(* IEC 61131-3 sources: Simulated-machine/integrations/openplc/thermal-plant-v4/pous/programs, 1 file *)

(* ---- main.st ---- *)
(* Generated by tools/generate_openplc_gateway.py.
   Raw Modbus values are intentionally retained; engineering_value = raw / scale.
   The cyclic task interval is 20 ms. *)
PROGRAM main
  VAR
    i_watchdog_scan_count : UINT := 0;
    i_watchdog_tick : BOOL := FALSE;
    i_condenser_last_echo : UINT := 0;
    i_condenser_echo_stale_ticks : UINT := 0;
    i_condenser_comm_lost : BOOL := FALSE;
    i_condensate_pump_last_echo : UINT := 0;
    i_condensate_pump_echo_stale_ticks : UINT := 0;
    i_condensate_pump_comm_lost : BOOL := FALSE;
    i_feedwater_tank_last_echo : UINT := 0;
    i_feedwater_tank_echo_stale_ticks : UINT := 0;
    i_feedwater_tank_comm_lost : BOOL := FALSE;
    i_feedwater_pump_last_echo : UINT := 0;
    i_feedwater_pump_echo_stale_ticks : UINT := 0;
    i_feedwater_pump_comm_lost : BOOL := FALSE;
    i_boiler_last_echo : UINT := 0;
    i_boiler_echo_stale_ticks : UINT := 0;
    i_boiler_comm_lost : BOOL := FALSE;
    i_steam_valve_last_echo : UINT := 0;
    i_steam_valve_echo_stale_ticks : UINT := 0;
    i_steam_valve_comm_lost : BOOL := FALSE;
    i_turbine_last_echo : UINT := 0;
    i_turbine_echo_stale_ticks : UINT := 0;
    i_turbine_comm_lost : BOOL := FALSE;
    i_generator_last_echo : UINT := 0;
    i_generator_echo_stale_ticks : UINT := 0;
    i_generator_comm_lost : BOOL := FALSE;
    i_condenser_start_active : BOOL := FALSE;
    i_condenser_start_scans : UINT := 0;
    i_condenser_stop_active : BOOL := FALSE;
    i_condenser_stop_scans : UINT := 0;
    i_condenser_reset_trip_active : BOOL := FALSE;
    i_condenser_reset_trip_scans : UINT := 0;
    i_condenser_ack_alarm_active : BOOL := FALSE;
    i_condenser_ack_alarm_scans : UINT := 0;
    i_condenser_trip_test_active : BOOL := FALSE;
    i_condenser_trip_test_scans : UINT := 0;
    i_condenser_clear_totalizer_active : BOOL := FALSE;
    i_condenser_clear_totalizer_scans : UINT := 0;
    i_condensate_pump_start_active : BOOL := FALSE;
    i_condensate_pump_start_scans : UINT := 0;
    i_condensate_pump_stop_active : BOOL := FALSE;
    i_condensate_pump_stop_scans : UINT := 0;
    i_condensate_pump_reset_trip_active : BOOL := FALSE;
    i_condensate_pump_reset_trip_scans : UINT := 0;
    i_condensate_pump_ack_alarm_active : BOOL := FALSE;
    i_condensate_pump_ack_alarm_scans : UINT := 0;
    i_condensate_pump_trip_test_active : BOOL := FALSE;
    i_condensate_pump_trip_test_scans : UINT := 0;
    i_condensate_pump_clear_totalizer_active : BOOL := FALSE;
    i_condensate_pump_clear_totalizer_scans : UINT := 0;
    i_feedwater_tank_start_active : BOOL := FALSE;
    i_feedwater_tank_start_scans : UINT := 0;
    i_feedwater_tank_stop_active : BOOL := FALSE;
    i_feedwater_tank_stop_scans : UINT := 0;
    i_feedwater_tank_reset_trip_active : BOOL := FALSE;
    i_feedwater_tank_reset_trip_scans : UINT := 0;
    i_feedwater_tank_ack_alarm_active : BOOL := FALSE;
    i_feedwater_tank_ack_alarm_scans : UINT := 0;
    i_feedwater_tank_trip_test_active : BOOL := FALSE;
    i_feedwater_tank_trip_test_scans : UINT := 0;
    i_feedwater_tank_clear_totalizer_active : BOOL := FALSE;
    i_feedwater_tank_clear_totalizer_scans : UINT := 0;
    i_feedwater_pump_start_active : BOOL := FALSE;
    i_feedwater_pump_start_scans : UINT := 0;
    i_feedwater_pump_stop_active : BOOL := FALSE;
    i_feedwater_pump_stop_scans : UINT := 0;
    i_feedwater_pump_reset_trip_active : BOOL := FALSE;
    i_feedwater_pump_reset_trip_scans : UINT := 0;
    i_feedwater_pump_ack_alarm_active : BOOL := FALSE;
    i_feedwater_pump_ack_alarm_scans : UINT := 0;
    i_feedwater_pump_trip_test_active : BOOL := FALSE;
    i_feedwater_pump_trip_test_scans : UINT := 0;
    i_feedwater_pump_clear_totalizer_active : BOOL := FALSE;
    i_feedwater_pump_clear_totalizer_scans : UINT := 0;
    i_boiler_start_active : BOOL := FALSE;
    i_boiler_start_scans : UINT := 0;
    i_boiler_stop_active : BOOL := FALSE;
    i_boiler_stop_scans : UINT := 0;
    i_boiler_reset_trip_active : BOOL := FALSE;
    i_boiler_reset_trip_scans : UINT := 0;
    i_boiler_ack_alarm_active : BOOL := FALSE;
    i_boiler_ack_alarm_scans : UINT := 0;
    i_boiler_trip_test_active : BOOL := FALSE;
    i_boiler_trip_test_scans : UINT := 0;
    i_boiler_clear_totalizer_active : BOOL := FALSE;
    i_boiler_clear_totalizer_scans : UINT := 0;
    i_steam_valve_start_active : BOOL := FALSE;
    i_steam_valve_start_scans : UINT := 0;
    i_steam_valve_stop_active : BOOL := FALSE;
    i_steam_valve_stop_scans : UINT := 0;
    i_steam_valve_reset_trip_active : BOOL := FALSE;
    i_steam_valve_reset_trip_scans : UINT := 0;
    i_steam_valve_ack_alarm_active : BOOL := FALSE;
    i_steam_valve_ack_alarm_scans : UINT := 0;
    i_steam_valve_trip_test_active : BOOL := FALSE;
    i_steam_valve_trip_test_scans : UINT := 0;
    i_steam_valve_clear_totalizer_active : BOOL := FALSE;
    i_steam_valve_clear_totalizer_scans : UINT := 0;
    i_turbine_start_active : BOOL := FALSE;
    i_turbine_start_scans : UINT := 0;
    i_turbine_stop_active : BOOL := FALSE;
    i_turbine_stop_scans : UINT := 0;
    i_turbine_reset_trip_active : BOOL := FALSE;
    i_turbine_reset_trip_scans : UINT := 0;
    i_turbine_ack_alarm_active : BOOL := FALSE;
    i_turbine_ack_alarm_scans : UINT := 0;
    i_turbine_trip_test_active : BOOL := FALSE;
    i_turbine_trip_test_scans : UINT := 0;
    i_turbine_clear_totalizer_active : BOOL := FALSE;
    i_turbine_clear_totalizer_scans : UINT := 0;
    i_generator_start_active : BOOL := FALSE;
    i_generator_start_scans : UINT := 0;
    i_generator_stop_active : BOOL := FALSE;
    i_generator_stop_scans : UINT := 0;
    i_generator_reset_trip_active : BOOL := FALSE;
    i_generator_reset_trip_scans : UINT := 0;
    i_generator_ack_alarm_active : BOOL := FALSE;
    i_generator_ack_alarm_scans : UINT := 0;
    i_generator_trip_test_active : BOOL := FALSE;
    i_generator_trip_test_scans : UINT := 0;
    i_generator_clear_totalizer_active : BOOL := FALSE;
    i_generator_clear_totalizer_scans : UINT := 0;
    i_generator_breaker_close_active : BOOL := FALSE;
    i_generator_breaker_close_scans : UINT := 0;
    i_generator_breaker_open_active : BOOL := FALSE;
    i_generator_breaker_open_scans : UINT := 0;
    i_turbine_trip_prev : BOOL := FALSE;
    i_boiler_trip_prev : BOOL := FALSE;
    i_condenser_trip_prev : BOOL := FALSE;
    i_feedwater_pump_trip_prev : BOOL := FALSE;
    i_condensate_pump_trip_prev : BOOL := FALSE;
    i_steam_valve_trip_prev : BOOL := FALSE;

    (* Southbound mirrors and commands.  Aliases match remote JSON exactly. *)
    condenser__input__status_word AT %IW0 : UINT := 0;
    condenser__input__alarm_word_1 AT %IW1 : UINT := 0;
    condenser__input__alarm_word_2 AT %IW2 : UINT := 0;
    condenser__input__trip_word AT %IW3 : UINT := 0;
    condenser__input__device_state AT %IW4 : UINT := 0;
    condenser__input__first_out_code AT %IW5 : UINT := 0;
    condenser__input__overall_quality AT %IW6 : UINT := 0;
    condenser__input__register_map_version AT %IW7 : UINT := 0;
    condenser__input__firmware_version AT %IW8 : UINT := 0;
    condenser__input__condenser_pressure AT %IW9 : UINT := 0;
    condenser__input__vacuum AT %IW10 : UINT := 0;
    condenser__input__hotwell_level AT %IW11 : UINT := 0;
    condenser__input__exhaust_inflow AT %IW12 : UINT := 0;
    condenser__input__condensing_capacity AT %IW13 : UINT := 0;
    condenser__input__actual_condensed AT %IW14 : UINT := 0;
    condenser__input__condensate_outflow AT %IW15 : UINT := 0;
    condenser__input__cooling_water_availability AT %IW16 : UINT := 0;
    condenser__input__vacuum_system_output AT %IW17 : UINT := 0;
    condenser__input__condensate_temperature AT %IW18 : UINT := 0;
    condenser__input__hotwell_mass_hi AT %IW19 : UINT := 0;
    condenser__input__hotwell_mass_lo AT %IW20 : UINT := 0;
    condenser__input__reserved_21 AT %IW21 : UINT := 0;
    condenser__input__reserved_22 AT %IW22 : UINT := 0;
    condenser__input__reserved_23 AT %IW23 : UINT := 0;
    condenser__input__reserved_24 AT %IW24 : UINT := 0;
    condenser__input__reserved_25 AT %IW25 : UINT := 0;
    condenser__input__reserved_26 AT %IW26 : UINT := 0;
    condenser__input__reserved_27 AT %IW27 : UINT := 0;
    condenser__input__reserved_28 AT %IW28 : UINT := 0;
    condenser__input__watchdog_echo AT %IW29 : UINT := 0;
    condenser__input__scan_time_ms AT %IW30 : UINT := 0;
    condenser__input__modbus_request_count AT %IW31 : UINT := 0;
    condenser__input__rejected_command_count AT %IW32 : UINT := 0;
    condenser__input__exception_count AT %IW33 : UINT := 0;
    condenser__input__sim_quality_word AT %IW34 : UINT := 0;
    condenser__input__sim_tick_low AT %IW35 : UINT := 0;
    condenser__input__comm_loss_seconds AT %IW36 : UINT := 0;
    condenser__input__fault_inject_word AT %IW37 : UINT := 0;
    condenser__input__snapshot_generation AT %IW38 : UINT := 0;
    condenser__input__run_seconds_hi AT %IW39 : UINT := 0;
    condenser__input__run_seconds_lo AT %IW40 : UINT := 0;
    condenser__input__start_count AT %IW41 : UINT := 0;
    condenser__input__trip_count AT %IW42 : UINT := 0;
    condenser__input__mass_total_hi AT %IW43 : UINT := 0;
    condenser__input__mass_total_lo AT %IW44 : UINT := 0;
    condenser__input__energy_total_hi AT %IW45 : UINT := 0;
    condenser__input__energy_total_lo AT %IW46 : UINT := 0;
    condenser__input__alarm_count AT %IW47 : UINT := 0;
    condenser__input__accepted_command_count AT %IW48 : UINT := 0;
    condenser__input__reserved_49 AT %IW49 : UINT := 0;
    condenser__discrete__ready AT %IX0.0 : BOOL := FALSE;
    condenser__discrete__running AT %IX0.1 : BOOL := FALSE;
    condenser__discrete__starting AT %IX0.2 : BOOL := FALSE;
    condenser__discrete__stopping AT %IX0.3 : BOOL := FALSE;
    condenser__discrete__tripped AT %IX0.4 : BOOL := FALSE;
    condenser__discrete__alarm_active AT %IX0.5 : BOOL := FALSE;
    condenser__discrete__local_mode AT %IX0.6 : BOOL := FALSE;
    condenser__discrete__remote_mode AT %IX0.7 : BOOL := FALSE;
    condenser__discrete__auto_mode AT %IX1.0 : BOOL := FALSE;
    condenser__discrete__manual_mode AT %IX1.1 : BOOL := FALSE;
    condenser__discrete__control_watchdog_ok AT %IX1.2 : BOOL := FALSE;
    condenser__discrete__sim_bus_ok AT %IX1.3 : BOOL := FALSE;
    condenser__discrete__interlocks_ok AT %IX1.4 : BOOL := FALSE;
    condenser__discrete__sensor_fault AT %IX1.5 : BOOL := FALSE;
    condenser__discrete__actuator_fault AT %IX1.6 : BOOL := FALSE;
    condenser__discrete__maintenance_mode AT %IX1.7 : BOOL := FALSE;
    condenser__holding_readback__control_mode AT %IW512 : UINT := 0;
    condenser__holding_readback__command_sequence AT %IW513 : UINT := 0;
    condenser__holding_readback__watchdog_counter AT %IW514 : UINT := 0;
    condenser__holding_readback__reset_key AT %IW515 : UINT := 0;
    condenser__holding_readback__simulation_flags AT %IW516 : UINT := 0;
    condenser__holding_readback__active_controller_id AT %IW517 : UINT := 0;
    condenser__holding_readback__command_lease_time AT %IW518 : UINT := 0;
    condenser__holding_readback__output_rate_limit AT %IW519 : UINT := 0;
    condenser__holding_readback__reserved AT %IW520 : UINT := 0;
    condenser__holding_readback__primary_setpoint AT %IW521 : UINT := 0;
    condenser__holding_readback__secondary_setpoint AT %IW522 : UINT := 0;
    condenser__holding_readback__manual_output AT %IW523 : UINT := 0;
    condenser__holding_readback__output_high_limit AT %IW524 : UINT := 0;
    condenser__holding_readback__output_low_limit AT %IW525 : UINT := 0;
    condenser__holding_readback__reserved_14 AT %IW526 : UINT := 0;
    condenser__holding_readback__reserved_15 AT %IW527 : UINT := 0;
    condenser__holding_readback__reserved_16 AT %IW528 : UINT := 0;
    condenser__holding_readback__reserved_17 AT %IW529 : UINT := 0;
    condenser__holding_readback__reserved_18 AT %IW530 : UINT := 0;
    condenser__holding_readback__pid_kp AT %IW531 : UINT := 0;
    condenser__holding_readback__pid_ki AT %IW532 : UINT := 0;
    condenser__holding_readback__pid_kd AT %IW533 : UINT := 0;
    condenser__holding_readback__deadband AT %IW534 : UINT := 0;
    condenser__holding_readback__integral_limit AT %IW535 : UINT := 0;
    condenser__holding_readback__controller_scan_time AT %IW536 : UINT := 0;
    condenser__holding_readback__reserved_25 AT %IW537 : UINT := 0;
    condenser__holding_readback__reserved_26 AT %IW538 : UINT := 0;
    condenser__holding_readback__reserved_27 AT %IW539 : UINT := 0;
    condenser__holding_readback__reserved_28 AT %IW540 : UINT := 0;
    condenser__holding_readback__makeup_valve_cmd AT %IW541 : UINT := 0;
    condenser__holding_readback__reserved_30 AT %IW542 : UINT := 0;
    condenser__holding_readback__reserved_31 AT %IW543 : UINT := 0;
    condenser__coil__start AT %QX0.0 : BOOL := FALSE;
    condenser__coil__stop AT %QX0.1 : BOOL := FALSE;
    condenser__coil__reset_trip AT %QX0.2 : BOOL := FALSE;
    condenser__coil__ack_alarm AT %QX0.3 : BOOL := FALSE;
    condenser__coil__emergency_stop AT %QX0.4 : BOOL := FALSE;
    condenser__coil__force_safe AT %QX0.5 : BOOL := FALSE;
    condenser__coil__trip_test AT %QX0.6 : BOOL := FALSE;
    condenser__coil__clear_totalizer AT %QX0.7 : BOOL := FALSE;
    condenser__holding__control_mode AT %QW0 : UINT := 3;
    condenser__holding__command_sequence AT %QW1 : UINT := 0;
    condenser__holding__watchdog_counter AT %QW2 : UINT := 1;
    condenser__holding__reset_key AT %QW3 : UINT := 0;
    condenser__holding__simulation_flags AT %QW4 : UINT := 0;
    condenser__holding__active_controller_id AT %QW5 : UINT := 1;
    condenser__holding__command_lease_time AT %QW6 : UINT := 5;
    condenser__holding__output_rate_limit AT %QW7 : UINT := 1000;
    condenser__holding__reserved AT %QW8 : UINT := 0;
    condenser__holding__primary_setpoint AT %QW9 : UINT := 0;
    condenser__holding__secondary_setpoint AT %QW10 : UINT := 0;
    condenser__holding__manual_output AT %QW11 : UINT := 0;
    condenser__holding__output_high_limit AT %QW12 : UINT := 10000;
    condenser__holding__output_low_limit AT %QW13 : UINT := 0;
    condenser__holding__pid_kp AT %QW19 : UINT := 0;
    condenser__holding__pid_ki AT %QW20 : UINT := 0;
    condenser__holding__pid_kd AT %QW21 : UINT := 0;
    condenser__holding__deadband AT %QW22 : UINT := 0;
    condenser__holding__integral_limit AT %QW23 : UINT := 0;
    condenser__holding__controller_scan_time AT %QW24 : UINT := 200;
    condenser__holding__makeup_valve_cmd AT %QW29 : UINT := 0;
    condensate_pump__input__status_word AT %IW64 : UINT := 0;
    condensate_pump__input__alarm_word_1 AT %IW65 : UINT := 0;
    condensate_pump__input__alarm_word_2 AT %IW66 : UINT := 0;
    condensate_pump__input__trip_word AT %IW67 : UINT := 0;
    condensate_pump__input__device_state AT %IW68 : UINT := 0;
    condensate_pump__input__first_out_code AT %IW69 : UINT := 0;
    condensate_pump__input__overall_quality AT %IW70 : UINT := 0;
    condensate_pump__input__register_map_version AT %IW71 : UINT := 0;
    condensate_pump__input__firmware_version AT %IW72 : UINT := 0;
    condensate_pump__input__actual_speed AT %IW73 : UINT := 0;
    condensate_pump__input__flow AT %IW74 : UINT := 0;
    condensate_pump__input__suction_pressure AT %IW75 : UINT := 0;
    condensate_pump__input__discharge_pressure AT %IW76 : UINT := 0;
    condensate_pump__input__motor_current AT %IW77 : UINT := 0;
    condensate_pump__input__npsh_margin AT %IW78 : UINT := 0;
    condensate_pump__input__vibration AT %IW79 : UINT := 0;
    condensate_pump__input__source_level AT %IW80 : UINT := 0;
    condensate_pump__input__backpressure AT %IW81 : UINT := 0;
    condensate_pump__input__outlet_valve_position AT %IW82 : UINT := 0;
    condensate_pump__input__cavitation_factor AT %IW83 : UINT := 0;
    condensate_pump__input__reserved_20 AT %IW84 : UINT := 0;
    condensate_pump__input__reserved_21 AT %IW85 : UINT := 0;
    condensate_pump__input__reserved_22 AT %IW86 : UINT := 0;
    condensate_pump__input__reserved_23 AT %IW87 : UINT := 0;
    condensate_pump__input__reserved_24 AT %IW88 : UINT := 0;
    condensate_pump__input__reserved_25 AT %IW89 : UINT := 0;
    condensate_pump__input__reserved_26 AT %IW90 : UINT := 0;
    condensate_pump__input__reserved_27 AT %IW91 : UINT := 0;
    condensate_pump__input__reserved_28 AT %IW92 : UINT := 0;
    condensate_pump__input__watchdog_echo AT %IW93 : UINT := 0;
    condensate_pump__input__scan_time_ms AT %IW94 : UINT := 0;
    condensate_pump__input__modbus_request_count AT %IW95 : UINT := 0;
    condensate_pump__input__rejected_command_count AT %IW96 : UINT := 0;
    condensate_pump__input__exception_count AT %IW97 : UINT := 0;
    condensate_pump__input__sim_quality_word AT %IW98 : UINT := 0;
    condensate_pump__input__sim_tick_low AT %IW99 : UINT := 0;
    condensate_pump__input__comm_loss_seconds AT %IW100 : UINT := 0;
    condensate_pump__input__fault_inject_word AT %IW101 : UINT := 0;
    condensate_pump__input__snapshot_generation AT %IW102 : UINT := 0;
    condensate_pump__input__run_seconds_hi AT %IW103 : UINT := 0;
    condensate_pump__input__run_seconds_lo AT %IW104 : UINT := 0;
    condensate_pump__input__start_count AT %IW105 : UINT := 0;
    condensate_pump__input__trip_count AT %IW106 : UINT := 0;
    condensate_pump__input__mass_total_hi AT %IW107 : UINT := 0;
    condensate_pump__input__mass_total_lo AT %IW108 : UINT := 0;
    condensate_pump__input__energy_total_hi AT %IW109 : UINT := 0;
    condensate_pump__input__energy_total_lo AT %IW110 : UINT := 0;
    condensate_pump__input__alarm_count AT %IW111 : UINT := 0;
    condensate_pump__input__accepted_command_count AT %IW112 : UINT := 0;
    condensate_pump__input__reserved_49 AT %IW113 : UINT := 0;
    condensate_pump__discrete__ready AT %IX2.0 : BOOL := FALSE;
    condensate_pump__discrete__running AT %IX2.1 : BOOL := FALSE;
    condensate_pump__discrete__starting AT %IX2.2 : BOOL := FALSE;
    condensate_pump__discrete__stopping AT %IX2.3 : BOOL := FALSE;
    condensate_pump__discrete__tripped AT %IX2.4 : BOOL := FALSE;
    condensate_pump__discrete__alarm_active AT %IX2.5 : BOOL := FALSE;
    condensate_pump__discrete__local_mode AT %IX2.6 : BOOL := FALSE;
    condensate_pump__discrete__remote_mode AT %IX2.7 : BOOL := FALSE;
    condensate_pump__discrete__auto_mode AT %IX3.0 : BOOL := FALSE;
    condensate_pump__discrete__manual_mode AT %IX3.1 : BOOL := FALSE;
    condensate_pump__discrete__control_watchdog_ok AT %IX3.2 : BOOL := FALSE;
    condensate_pump__discrete__sim_bus_ok AT %IX3.3 : BOOL := FALSE;
    condensate_pump__discrete__interlocks_ok AT %IX3.4 : BOOL := FALSE;
    condensate_pump__discrete__sensor_fault AT %IX3.5 : BOOL := FALSE;
    condensate_pump__discrete__actuator_fault AT %IX3.6 : BOOL := FALSE;
    condensate_pump__discrete__maintenance_mode AT %IX3.7 : BOOL := FALSE;
    condensate_pump__holding_readback__control_mode AT %IW576 : UINT := 0;
    condensate_pump__holding_readback__command_sequence AT %IW577 : UINT := 0;
    condensate_pump__holding_readback__watchdog_counter AT %IW578 : UINT := 0;
    condensate_pump__holding_readback__reset_key AT %IW579 : UINT := 0;
    condensate_pump__holding_readback__simulation_flags AT %IW580 : UINT := 0;
    condensate_pump__holding_readback__active_controller_id AT %IW581 : UINT := 0;
    condensate_pump__holding_readback__command_lease_time AT %IW582 : UINT := 0;
    condensate_pump__holding_readback__output_rate_limit AT %IW583 : UINT := 0;
    condensate_pump__holding_readback__reserved AT %IW584 : UINT := 0;
    condensate_pump__holding_readback__primary_setpoint AT %IW585 : UINT := 0;
    condensate_pump__holding_readback__secondary_setpoint AT %IW586 : UINT := 0;
    condensate_pump__holding_readback__manual_output AT %IW587 : UINT := 0;
    condensate_pump__holding_readback__output_high_limit AT %IW588 : UINT := 0;
    condensate_pump__holding_readback__output_low_limit AT %IW589 : UINT := 0;
    condensate_pump__holding_readback__reserved_14 AT %IW590 : UINT := 0;
    condensate_pump__holding_readback__reserved_15 AT %IW591 : UINT := 0;
    condensate_pump__holding_readback__reserved_16 AT %IW592 : UINT := 0;
    condensate_pump__holding_readback__reserved_17 AT %IW593 : UINT := 0;
    condensate_pump__holding_readback__reserved_18 AT %IW594 : UINT := 0;
    condensate_pump__holding_readback__pid_kp AT %IW595 : UINT := 0;
    condensate_pump__holding_readback__pid_ki AT %IW596 : UINT := 0;
    condensate_pump__holding_readback__pid_kd AT %IW597 : UINT := 0;
    condensate_pump__holding_readback__deadband AT %IW598 : UINT := 0;
    condensate_pump__holding_readback__integral_limit AT %IW599 : UINT := 0;
    condensate_pump__holding_readback__controller_scan_time AT %IW600 : UINT := 0;
    condensate_pump__holding_readback__reserved_25 AT %IW601 : UINT := 0;
    condensate_pump__holding_readback__reserved_26 AT %IW602 : UINT := 0;
    condensate_pump__holding_readback__reserved_27 AT %IW603 : UINT := 0;
    condensate_pump__holding_readback__reserved_28 AT %IW604 : UINT := 0;
    condensate_pump__holding_readback__reserved_29 AT %IW605 : UINT := 0;
    condensate_pump__holding_readback__reserved_30 AT %IW606 : UINT := 0;
    condensate_pump__holding_readback__reserved_31 AT %IW607 : UINT := 0;
    condensate_pump__coil__start AT %QX2.0 : BOOL := FALSE;
    condensate_pump__coil__stop AT %QX2.1 : BOOL := FALSE;
    condensate_pump__coil__reset_trip AT %QX2.2 : BOOL := FALSE;
    condensate_pump__coil__ack_alarm AT %QX2.3 : BOOL := FALSE;
    condensate_pump__coil__emergency_stop AT %QX2.4 : BOOL := FALSE;
    condensate_pump__coil__force_safe AT %QX2.5 : BOOL := FALSE;
    condensate_pump__coil__trip_test AT %QX2.6 : BOOL := FALSE;
    condensate_pump__coil__clear_totalizer AT %QX2.7 : BOOL := FALSE;
    condensate_pump__holding__control_mode AT %QW64 : UINT := 3;
    condensate_pump__holding__command_sequence AT %QW65 : UINT := 0;
    condensate_pump__holding__watchdog_counter AT %QW66 : UINT := 1;
    condensate_pump__holding__reset_key AT %QW67 : UINT := 0;
    condensate_pump__holding__simulation_flags AT %QW68 : UINT := 0;
    condensate_pump__holding__active_controller_id AT %QW69 : UINT := 2;
    condensate_pump__holding__command_lease_time AT %QW70 : UINT := 5;
    condensate_pump__holding__output_rate_limit AT %QW71 : UINT := 1000;
    condensate_pump__holding__reserved AT %QW72 : UINT := 0;
    condensate_pump__holding__primary_setpoint AT %QW73 : UINT := 0;
    condensate_pump__holding__secondary_setpoint AT %QW74 : UINT := 0;
    condensate_pump__holding__manual_output AT %QW75 : UINT := 0;
    condensate_pump__holding__output_high_limit AT %QW76 : UINT := 10000;
    condensate_pump__holding__output_low_limit AT %QW77 : UINT := 0;
    condensate_pump__holding__pid_kp AT %QW83 : UINT := 0;
    condensate_pump__holding__pid_ki AT %QW84 : UINT := 0;
    condensate_pump__holding__pid_kd AT %QW85 : UINT := 0;
    condensate_pump__holding__deadband AT %QW86 : UINT := 0;
    condensate_pump__holding__integral_limit AT %QW87 : UINT := 0;
    condensate_pump__holding__controller_scan_time AT %QW88 : UINT := 200;
    feedwater_tank__input__status_word AT %IW128 : UINT := 0;
    feedwater_tank__input__alarm_word_1 AT %IW129 : UINT := 0;
    feedwater_tank__input__alarm_word_2 AT %IW130 : UINT := 0;
    feedwater_tank__input__trip_word AT %IW131 : UINT := 0;
    feedwater_tank__input__device_state AT %IW132 : UINT := 0;
    feedwater_tank__input__first_out_code AT %IW133 : UINT := 0;
    feedwater_tank__input__overall_quality AT %IW134 : UINT := 0;
    feedwater_tank__input__register_map_version AT %IW135 : UINT := 0;
    feedwater_tank__input__firmware_version AT %IW136 : UINT := 0;
    feedwater_tank__input__tank_level AT %IW137 : UINT := 0;
    feedwater_tank__input__tank_mass_hi AT %IW138 : UINT := 0;
    feedwater_tank__input__tank_mass_lo AT %IW139 : UINT := 0;
    feedwater_tank__input__condensate_inflow AT %IW140 : UINT := 0;
    feedwater_tank__input__feedwater_outflow AT %IW141 : UINT := 0;
    feedwater_tank__input__water_temperature AT %IW142 : UINT := 0;
    feedwater_tank__input__tank_pressure AT %IW143 : UINT := 0;
    feedwater_tank__input__overflow_flow AT %IW144 : UINT := 0;
    feedwater_tank__input__net_flow AT %IW145 : UINT := 0;
    feedwater_tank__input__reserved_18 AT %IW146 : UINT := 0;
    feedwater_tank__input__reserved_19 AT %IW147 : UINT := 0;
    feedwater_tank__input__reserved_20 AT %IW148 : UINT := 0;
    feedwater_tank__input__reserved_21 AT %IW149 : UINT := 0;
    feedwater_tank__input__reserved_22 AT %IW150 : UINT := 0;
    feedwater_tank__input__reserved_23 AT %IW151 : UINT := 0;
    feedwater_tank__input__reserved_24 AT %IW152 : UINT := 0;
    feedwater_tank__input__reserved_25 AT %IW153 : UINT := 0;
    feedwater_tank__input__reserved_26 AT %IW154 : UINT := 0;
    feedwater_tank__input__reserved_27 AT %IW155 : UINT := 0;
    feedwater_tank__input__reserved_28 AT %IW156 : UINT := 0;
    feedwater_tank__input__watchdog_echo AT %IW157 : UINT := 0;
    feedwater_tank__input__scan_time_ms AT %IW158 : UINT := 0;
    feedwater_tank__input__modbus_request_count AT %IW159 : UINT := 0;
    feedwater_tank__input__rejected_command_count AT %IW160 : UINT := 0;
    feedwater_tank__input__exception_count AT %IW161 : UINT := 0;
    feedwater_tank__input__sim_quality_word AT %IW162 : UINT := 0;
    feedwater_tank__input__sim_tick_low AT %IW163 : UINT := 0;
    feedwater_tank__input__comm_loss_seconds AT %IW164 : UINT := 0;
    feedwater_tank__input__fault_inject_word AT %IW165 : UINT := 0;
    feedwater_tank__input__snapshot_generation AT %IW166 : UINT := 0;
    feedwater_tank__input__run_seconds_hi AT %IW167 : UINT := 0;
    feedwater_tank__input__run_seconds_lo AT %IW168 : UINT := 0;
    feedwater_tank__input__start_count AT %IW169 : UINT := 0;
    feedwater_tank__input__trip_count AT %IW170 : UINT := 0;
    feedwater_tank__input__mass_total_hi AT %IW171 : UINT := 0;
    feedwater_tank__input__mass_total_lo AT %IW172 : UINT := 0;
    feedwater_tank__input__energy_total_hi AT %IW173 : UINT := 0;
    feedwater_tank__input__energy_total_lo AT %IW174 : UINT := 0;
    feedwater_tank__input__alarm_count AT %IW175 : UINT := 0;
    feedwater_tank__input__accepted_command_count AT %IW176 : UINT := 0;
    feedwater_tank__input__reserved_49 AT %IW177 : UINT := 0;
    feedwater_tank__discrete__ready AT %IX4.0 : BOOL := FALSE;
    feedwater_tank__discrete__running AT %IX4.1 : BOOL := FALSE;
    feedwater_tank__discrete__starting AT %IX4.2 : BOOL := FALSE;
    feedwater_tank__discrete__stopping AT %IX4.3 : BOOL := FALSE;
    feedwater_tank__discrete__tripped AT %IX4.4 : BOOL := FALSE;
    feedwater_tank__discrete__alarm_active AT %IX4.5 : BOOL := FALSE;
    feedwater_tank__discrete__local_mode AT %IX4.6 : BOOL := FALSE;
    feedwater_tank__discrete__remote_mode AT %IX4.7 : BOOL := FALSE;
    feedwater_tank__discrete__auto_mode AT %IX5.0 : BOOL := FALSE;
    feedwater_tank__discrete__manual_mode AT %IX5.1 : BOOL := FALSE;
    feedwater_tank__discrete__control_watchdog_ok AT %IX5.2 : BOOL := FALSE;
    feedwater_tank__discrete__sim_bus_ok AT %IX5.3 : BOOL := FALSE;
    feedwater_tank__discrete__interlocks_ok AT %IX5.4 : BOOL := FALSE;
    feedwater_tank__discrete__sensor_fault AT %IX5.5 : BOOL := FALSE;
    feedwater_tank__discrete__actuator_fault AT %IX5.6 : BOOL := FALSE;
    feedwater_tank__discrete__maintenance_mode AT %IX5.7 : BOOL := FALSE;
    feedwater_tank__holding_readback__control_mode AT %IW640 : UINT := 0;
    feedwater_tank__holding_readback__command_sequence AT %IW641 : UINT := 0;
    feedwater_tank__holding_readback__watchdog_counter AT %IW642 : UINT := 0;
    feedwater_tank__holding_readback__reset_key AT %IW643 : UINT := 0;
    feedwater_tank__holding_readback__simulation_flags AT %IW644 : UINT := 0;
    feedwater_tank__holding_readback__active_controller_id AT %IW645 : UINT := 0;
    feedwater_tank__holding_readback__command_lease_time AT %IW646 : UINT := 0;
    feedwater_tank__holding_readback__output_rate_limit AT %IW647 : UINT := 0;
    feedwater_tank__holding_readback__reserved AT %IW648 : UINT := 0;
    feedwater_tank__holding_readback__primary_setpoint AT %IW649 : UINT := 0;
    feedwater_tank__holding_readback__secondary_setpoint AT %IW650 : UINT := 0;
    feedwater_tank__holding_readback__manual_output AT %IW651 : UINT := 0;
    feedwater_tank__holding_readback__output_high_limit AT %IW652 : UINT := 0;
    feedwater_tank__holding_readback__output_low_limit AT %IW653 : UINT := 0;
    feedwater_tank__holding_readback__reserved_14 AT %IW654 : UINT := 0;
    feedwater_tank__holding_readback__reserved_15 AT %IW655 : UINT := 0;
    feedwater_tank__holding_readback__reserved_16 AT %IW656 : UINT := 0;
    feedwater_tank__holding_readback__reserved_17 AT %IW657 : UINT := 0;
    feedwater_tank__holding_readback__reserved_18 AT %IW658 : UINT := 0;
    feedwater_tank__holding_readback__pid_kp AT %IW659 : UINT := 0;
    feedwater_tank__holding_readback__pid_ki AT %IW660 : UINT := 0;
    feedwater_tank__holding_readback__pid_kd AT %IW661 : UINT := 0;
    feedwater_tank__holding_readback__deadband AT %IW662 : UINT := 0;
    feedwater_tank__holding_readback__integral_limit AT %IW663 : UINT := 0;
    feedwater_tank__holding_readback__controller_scan_time AT %IW664 : UINT := 0;
    feedwater_tank__holding_readback__reserved_25 AT %IW665 : UINT := 0;
    feedwater_tank__holding_readback__reserved_26 AT %IW666 : UINT := 0;
    feedwater_tank__holding_readback__reserved_27 AT %IW667 : UINT := 0;
    feedwater_tank__holding_readback__reserved_28 AT %IW668 : UINT := 0;
    feedwater_tank__holding_readback__heating_setpoint AT %IW669 : UINT := 0;
    feedwater_tank__holding_readback__reserved_30 AT %IW670 : UINT := 0;
    feedwater_tank__holding_readback__reserved_31 AT %IW671 : UINT := 0;
    feedwater_tank__coil__start AT %QX4.0 : BOOL := FALSE;
    feedwater_tank__coil__stop AT %QX4.1 : BOOL := FALSE;
    feedwater_tank__coil__reset_trip AT %QX4.2 : BOOL := FALSE;
    feedwater_tank__coil__ack_alarm AT %QX4.3 : BOOL := FALSE;
    feedwater_tank__coil__emergency_stop AT %QX4.4 : BOOL := FALSE;
    feedwater_tank__coil__force_safe AT %QX4.5 : BOOL := FALSE;
    feedwater_tank__coil__trip_test AT %QX4.6 : BOOL := FALSE;
    feedwater_tank__coil__clear_totalizer AT %QX4.7 : BOOL := FALSE;
    feedwater_tank__holding__control_mode AT %QW128 : UINT := 3;
    feedwater_tank__holding__command_sequence AT %QW129 : UINT := 0;
    feedwater_tank__holding__watchdog_counter AT %QW130 : UINT := 1;
    feedwater_tank__holding__reset_key AT %QW131 : UINT := 0;
    feedwater_tank__holding__simulation_flags AT %QW132 : UINT := 0;
    feedwater_tank__holding__active_controller_id AT %QW133 : UINT := 3;
    feedwater_tank__holding__command_lease_time AT %QW134 : UINT := 5;
    feedwater_tank__holding__output_rate_limit AT %QW135 : UINT := 1000;
    feedwater_tank__holding__reserved AT %QW136 : UINT := 0;
    feedwater_tank__holding__primary_setpoint AT %QW137 : UINT := 0;
    feedwater_tank__holding__secondary_setpoint AT %QW138 : UINT := 0;
    feedwater_tank__holding__manual_output AT %QW139 : UINT := 0;
    feedwater_tank__holding__output_high_limit AT %QW140 : UINT := 10000;
    feedwater_tank__holding__output_low_limit AT %QW141 : UINT := 0;
    feedwater_tank__holding__pid_kp AT %QW147 : UINT := 0;
    feedwater_tank__holding__pid_ki AT %QW148 : UINT := 0;
    feedwater_tank__holding__pid_kd AT %QW149 : UINT := 0;
    feedwater_tank__holding__deadband AT %QW150 : UINT := 0;
    feedwater_tank__holding__integral_limit AT %QW151 : UINT := 0;
    feedwater_tank__holding__controller_scan_time AT %QW152 : UINT := 200;
    feedwater_tank__holding__heating_setpoint AT %QW157 : UINT := 200;
    feedwater_pump__input__status_word AT %IW192 : UINT := 0;
    feedwater_pump__input__alarm_word_1 AT %IW193 : UINT := 0;
    feedwater_pump__input__alarm_word_2 AT %IW194 : UINT := 0;
    feedwater_pump__input__trip_word AT %IW195 : UINT := 0;
    feedwater_pump__input__device_state AT %IW196 : UINT := 0;
    feedwater_pump__input__first_out_code AT %IW197 : UINT := 0;
    feedwater_pump__input__overall_quality AT %IW198 : UINT := 0;
    feedwater_pump__input__register_map_version AT %IW199 : UINT := 0;
    feedwater_pump__input__firmware_version AT %IW200 : UINT := 0;
    feedwater_pump__input__actual_speed AT %IW201 : UINT := 0;
    feedwater_pump__input__flow AT %IW202 : UINT := 0;
    feedwater_pump__input__suction_pressure AT %IW203 : UINT := 0;
    feedwater_pump__input__discharge_pressure AT %IW204 : UINT := 0;
    feedwater_pump__input__motor_current AT %IW205 : UINT := 0;
    feedwater_pump__input__npsh_margin AT %IW206 : UINT := 0;
    feedwater_pump__input__vibration AT %IW207 : UINT := 0;
    feedwater_pump__input__source_level AT %IW208 : UINT := 0;
    feedwater_pump__input__backpressure AT %IW209 : UINT := 0;
    feedwater_pump__input__outlet_valve_position AT %IW210 : UINT := 0;
    feedwater_pump__input__cavitation_factor AT %IW211 : UINT := 0;
    feedwater_pump__input__boiler_pressure AT %IW212 : UINT := 0;
    feedwater_pump__input__feedwater_permitted AT %IW213 : UINT := 0;
    feedwater_pump__input__reserved_22 AT %IW214 : UINT := 0;
    feedwater_pump__input__reserved_23 AT %IW215 : UINT := 0;
    feedwater_pump__input__reserved_24 AT %IW216 : UINT := 0;
    feedwater_pump__input__reserved_25 AT %IW217 : UINT := 0;
    feedwater_pump__input__reserved_26 AT %IW218 : UINT := 0;
    feedwater_pump__input__reserved_27 AT %IW219 : UINT := 0;
    feedwater_pump__input__reserved_28 AT %IW220 : UINT := 0;
    feedwater_pump__input__watchdog_echo AT %IW221 : UINT := 0;
    feedwater_pump__input__scan_time_ms AT %IW222 : UINT := 0;
    feedwater_pump__input__modbus_request_count AT %IW223 : UINT := 0;
    feedwater_pump__input__rejected_command_count AT %IW224 : UINT := 0;
    feedwater_pump__input__exception_count AT %IW225 : UINT := 0;
    feedwater_pump__input__sim_quality_word AT %IW226 : UINT := 0;
    feedwater_pump__input__sim_tick_low AT %IW227 : UINT := 0;
    feedwater_pump__input__comm_loss_seconds AT %IW228 : UINT := 0;
    feedwater_pump__input__fault_inject_word AT %IW229 : UINT := 0;
    feedwater_pump__input__snapshot_generation AT %IW230 : UINT := 0;
    feedwater_pump__input__run_seconds_hi AT %IW231 : UINT := 0;
    feedwater_pump__input__run_seconds_lo AT %IW232 : UINT := 0;
    feedwater_pump__input__start_count AT %IW233 : UINT := 0;
    feedwater_pump__input__trip_count AT %IW234 : UINT := 0;
    feedwater_pump__input__mass_total_hi AT %IW235 : UINT := 0;
    feedwater_pump__input__mass_total_lo AT %IW236 : UINT := 0;
    feedwater_pump__input__energy_total_hi AT %IW237 : UINT := 0;
    feedwater_pump__input__energy_total_lo AT %IW238 : UINT := 0;
    feedwater_pump__input__alarm_count AT %IW239 : UINT := 0;
    feedwater_pump__input__accepted_command_count AT %IW240 : UINT := 0;
    feedwater_pump__input__reserved_49 AT %IW241 : UINT := 0;
    feedwater_pump__discrete__ready AT %IX6.0 : BOOL := FALSE;
    feedwater_pump__discrete__running AT %IX6.1 : BOOL := FALSE;
    feedwater_pump__discrete__starting AT %IX6.2 : BOOL := FALSE;
    feedwater_pump__discrete__stopping AT %IX6.3 : BOOL := FALSE;
    feedwater_pump__discrete__tripped AT %IX6.4 : BOOL := FALSE;
    feedwater_pump__discrete__alarm_active AT %IX6.5 : BOOL := FALSE;
    feedwater_pump__discrete__local_mode AT %IX6.6 : BOOL := FALSE;
    feedwater_pump__discrete__remote_mode AT %IX6.7 : BOOL := FALSE;
    feedwater_pump__discrete__auto_mode AT %IX7.0 : BOOL := FALSE;
    feedwater_pump__discrete__manual_mode AT %IX7.1 : BOOL := FALSE;
    feedwater_pump__discrete__control_watchdog_ok AT %IX7.2 : BOOL := FALSE;
    feedwater_pump__discrete__sim_bus_ok AT %IX7.3 : BOOL := FALSE;
    feedwater_pump__discrete__interlocks_ok AT %IX7.4 : BOOL := FALSE;
    feedwater_pump__discrete__sensor_fault AT %IX7.5 : BOOL := FALSE;
    feedwater_pump__discrete__actuator_fault AT %IX7.6 : BOOL := FALSE;
    feedwater_pump__discrete__maintenance_mode AT %IX7.7 : BOOL := FALSE;
    feedwater_pump__holding_readback__control_mode AT %IW704 : UINT := 0;
    feedwater_pump__holding_readback__command_sequence AT %IW705 : UINT := 0;
    feedwater_pump__holding_readback__watchdog_counter AT %IW706 : UINT := 0;
    feedwater_pump__holding_readback__reset_key AT %IW707 : UINT := 0;
    feedwater_pump__holding_readback__simulation_flags AT %IW708 : UINT := 0;
    feedwater_pump__holding_readback__active_controller_id AT %IW709 : UINT := 0;
    feedwater_pump__holding_readback__command_lease_time AT %IW710 : UINT := 0;
    feedwater_pump__holding_readback__output_rate_limit AT %IW711 : UINT := 0;
    feedwater_pump__holding_readback__reserved AT %IW712 : UINT := 0;
    feedwater_pump__holding_readback__primary_setpoint AT %IW713 : UINT := 0;
    feedwater_pump__holding_readback__secondary_setpoint AT %IW714 : UINT := 0;
    feedwater_pump__holding_readback__manual_output AT %IW715 : UINT := 0;
    feedwater_pump__holding_readback__output_high_limit AT %IW716 : UINT := 0;
    feedwater_pump__holding_readback__output_low_limit AT %IW717 : UINT := 0;
    feedwater_pump__holding_readback__reserved_14 AT %IW718 : UINT := 0;
    feedwater_pump__holding_readback__reserved_15 AT %IW719 : UINT := 0;
    feedwater_pump__holding_readback__reserved_16 AT %IW720 : UINT := 0;
    feedwater_pump__holding_readback__reserved_17 AT %IW721 : UINT := 0;
    feedwater_pump__holding_readback__reserved_18 AT %IW722 : UINT := 0;
    feedwater_pump__holding_readback__pid_kp AT %IW723 : UINT := 0;
    feedwater_pump__holding_readback__pid_ki AT %IW724 : UINT := 0;
    feedwater_pump__holding_readback__pid_kd AT %IW725 : UINT := 0;
    feedwater_pump__holding_readback__deadband AT %IW726 : UINT := 0;
    feedwater_pump__holding_readback__integral_limit AT %IW727 : UINT := 0;
    feedwater_pump__holding_readback__controller_scan_time AT %IW728 : UINT := 0;
    feedwater_pump__holding_readback__reserved_25 AT %IW729 : UINT := 0;
    feedwater_pump__holding_readback__reserved_26 AT %IW730 : UINT := 0;
    feedwater_pump__holding_readback__reserved_27 AT %IW731 : UINT := 0;
    feedwater_pump__holding_readback__reserved_28 AT %IW732 : UINT := 0;
    feedwater_pump__holding_readback__outlet_valve_cmd AT %IW733 : UINT := 0;
    feedwater_pump__holding_readback__reserved_30 AT %IW734 : UINT := 0;
    feedwater_pump__holding_readback__reserved_31 AT %IW735 : UINT := 0;
    feedwater_pump__coil__start AT %QX6.0 : BOOL := FALSE;
    feedwater_pump__coil__stop AT %QX6.1 : BOOL := FALSE;
    feedwater_pump__coil__reset_trip AT %QX6.2 : BOOL := FALSE;
    feedwater_pump__coil__ack_alarm AT %QX6.3 : BOOL := FALSE;
    feedwater_pump__coil__emergency_stop AT %QX6.4 : BOOL := FALSE;
    feedwater_pump__coil__force_safe AT %QX6.5 : BOOL := FALSE;
    feedwater_pump__coil__trip_test AT %QX6.6 : BOOL := FALSE;
    feedwater_pump__coil__clear_totalizer AT %QX6.7 : BOOL := FALSE;
    feedwater_pump__holding__control_mode AT %QW192 : UINT := 3;
    feedwater_pump__holding__command_sequence AT %QW193 : UINT := 0;
    feedwater_pump__holding__watchdog_counter AT %QW194 : UINT := 1;
    feedwater_pump__holding__reset_key AT %QW195 : UINT := 0;
    feedwater_pump__holding__simulation_flags AT %QW196 : UINT := 0;
    feedwater_pump__holding__active_controller_id AT %QW197 : UINT := 4;
    feedwater_pump__holding__command_lease_time AT %QW198 : UINT := 5;
    feedwater_pump__holding__output_rate_limit AT %QW199 : UINT := 1000;
    feedwater_pump__holding__reserved AT %QW200 : UINT := 0;
    feedwater_pump__holding__primary_setpoint AT %QW201 : UINT := 0;
    feedwater_pump__holding__secondary_setpoint AT %QW202 : UINT := 0;
    feedwater_pump__holding__manual_output AT %QW203 : UINT := 0;
    feedwater_pump__holding__output_high_limit AT %QW204 : UINT := 10000;
    feedwater_pump__holding__output_low_limit AT %QW205 : UINT := 0;
    feedwater_pump__holding__pid_kp AT %QW211 : UINT := 0;
    feedwater_pump__holding__pid_ki AT %QW212 : UINT := 0;
    feedwater_pump__holding__pid_kd AT %QW213 : UINT := 0;
    feedwater_pump__holding__deadband AT %QW214 : UINT := 0;
    feedwater_pump__holding__integral_limit AT %QW215 : UINT := 0;
    feedwater_pump__holding__controller_scan_time AT %QW216 : UINT := 200;
    feedwater_pump__holding__outlet_valve_cmd AT %QW221 : UINT := 0;
    boiler__input__status_word AT %IW256 : UINT := 0;
    boiler__input__alarm_word_1 AT %IW257 : UINT := 0;
    boiler__input__alarm_word_2 AT %IW258 : UINT := 0;
    boiler__input__trip_word AT %IW259 : UINT := 0;
    boiler__input__device_state AT %IW260 : UINT := 0;
    boiler__input__first_out_code AT %IW261 : UINT := 0;
    boiler__input__overall_quality AT %IW262 : UINT := 0;
    boiler__input__register_map_version AT %IW263 : UINT := 0;
    boiler__input__firmware_version AT %IW264 : UINT := 0;
    boiler__input__boiler_pressure AT %IW265 : UINT := 0;
    boiler__input__level_indicated AT %IW266 : UINT := 0;
    boiler__input__level_actual AT %IW267 : UINT := 0;
    boiler__input__feedwater_flow AT %IW268 : UINT := 0;
    boiler__input__steam_generation AT %IW269 : UINT := 0;
    boiler__input__steam_outflow AT %IW270 : UINT := 0;
    boiler__input__burner_output AT %IW271 : UINT := 0;
    boiler__input__steam_temperature AT %IW272 : UINT := 0;
    boiler__input__water_mass_hi AT %IW273 : UINT := 0;
    boiler__input__water_mass_lo AT %IW274 : UINT := 0;
    boiler__input__flame_status AT %IW275 : UINT := 0;
    boiler__input__blowdown_flow AT %IW276 : UINT := 0;
    boiler__input__purge_time_remaining AT %IW277 : UINT := 0;
    boiler__input__feedwater_permitted AT %IW278 : UINT := 0;
    boiler__input__relief_flow AT %IW279 : UINT := 0;
    boiler__input__reserved_24 AT %IW280 : UINT := 0;
    boiler__input__reserved_25 AT %IW281 : UINT := 0;
    boiler__input__reserved_26 AT %IW282 : UINT := 0;
    boiler__input__reserved_27 AT %IW283 : UINT := 0;
    boiler__input__reserved_28 AT %IW284 : UINT := 0;
    boiler__input__watchdog_echo AT %IW285 : UINT := 0;
    boiler__input__scan_time_ms AT %IW286 : UINT := 0;
    boiler__input__modbus_request_count AT %IW287 : UINT := 0;
    boiler__input__rejected_command_count AT %IW288 : UINT := 0;
    boiler__input__exception_count AT %IW289 : UINT := 0;
    boiler__input__sim_quality_word AT %IW290 : UINT := 0;
    boiler__input__sim_tick_low AT %IW291 : UINT := 0;
    boiler__input__comm_loss_seconds AT %IW292 : UINT := 0;
    boiler__input__fault_inject_word AT %IW293 : UINT := 0;
    boiler__input__snapshot_generation AT %IW294 : UINT := 0;
    boiler__input__run_seconds_hi AT %IW295 : UINT := 0;
    boiler__input__run_seconds_lo AT %IW296 : UINT := 0;
    boiler__input__start_count AT %IW297 : UINT := 0;
    boiler__input__trip_count AT %IW298 : UINT := 0;
    boiler__input__mass_total_hi AT %IW299 : UINT := 0;
    boiler__input__mass_total_lo AT %IW300 : UINT := 0;
    boiler__input__energy_total_hi AT %IW301 : UINT := 0;
    boiler__input__energy_total_lo AT %IW302 : UINT := 0;
    boiler__input__alarm_count AT %IW303 : UINT := 0;
    boiler__input__accepted_command_count AT %IW304 : UINT := 0;
    boiler__input__reserved_49 AT %IW305 : UINT := 0;
    boiler__discrete__ready AT %IX8.0 : BOOL := FALSE;
    boiler__discrete__running AT %IX8.1 : BOOL := FALSE;
    boiler__discrete__starting AT %IX8.2 : BOOL := FALSE;
    boiler__discrete__stopping AT %IX8.3 : BOOL := FALSE;
    boiler__discrete__tripped AT %IX8.4 : BOOL := FALSE;
    boiler__discrete__alarm_active AT %IX8.5 : BOOL := FALSE;
    boiler__discrete__local_mode AT %IX8.6 : BOOL := FALSE;
    boiler__discrete__remote_mode AT %IX8.7 : BOOL := FALSE;
    boiler__discrete__auto_mode AT %IX9.0 : BOOL := FALSE;
    boiler__discrete__manual_mode AT %IX9.1 : BOOL := FALSE;
    boiler__discrete__control_watchdog_ok AT %IX9.2 : BOOL := FALSE;
    boiler__discrete__sim_bus_ok AT %IX9.3 : BOOL := FALSE;
    boiler__discrete__interlocks_ok AT %IX9.4 : BOOL := FALSE;
    boiler__discrete__sensor_fault AT %IX9.5 : BOOL := FALSE;
    boiler__discrete__actuator_fault AT %IX9.6 : BOOL := FALSE;
    boiler__discrete__maintenance_mode AT %IX9.7 : BOOL := FALSE;
    boiler__holding_readback__control_mode AT %IW768 : UINT := 0;
    boiler__holding_readback__command_sequence AT %IW769 : UINT := 0;
    boiler__holding_readback__watchdog_counter AT %IW770 : UINT := 0;
    boiler__holding_readback__reset_key AT %IW771 : UINT := 0;
    boiler__holding_readback__simulation_flags AT %IW772 : UINT := 0;
    boiler__holding_readback__active_controller_id AT %IW773 : UINT := 0;
    boiler__holding_readback__command_lease_time AT %IW774 : UINT := 0;
    boiler__holding_readback__output_rate_limit AT %IW775 : UINT := 0;
    boiler__holding_readback__reserved AT %IW776 : UINT := 0;
    boiler__holding_readback__primary_setpoint AT %IW777 : UINT := 0;
    boiler__holding_readback__secondary_setpoint AT %IW778 : UINT := 0;
    boiler__holding_readback__manual_output AT %IW779 : UINT := 0;
    boiler__holding_readback__output_high_limit AT %IW780 : UINT := 0;
    boiler__holding_readback__output_low_limit AT %IW781 : UINT := 0;
    boiler__holding_readback__reserved_14 AT %IW782 : UINT := 0;
    boiler__holding_readback__reserved_15 AT %IW783 : UINT := 0;
    boiler__holding_readback__reserved_16 AT %IW784 : UINT := 0;
    boiler__holding_readback__reserved_17 AT %IW785 : UINT := 0;
    boiler__holding_readback__reserved_18 AT %IW786 : UINT := 0;
    boiler__holding_readback__pid_kp AT %IW787 : UINT := 0;
    boiler__holding_readback__pid_ki AT %IW788 : UINT := 0;
    boiler__holding_readback__pid_kd AT %IW789 : UINT := 0;
    boiler__holding_readback__deadband AT %IW790 : UINT := 0;
    boiler__holding_readback__integral_limit AT %IW791 : UINT := 0;
    boiler__holding_readback__controller_scan_time AT %IW792 : UINT := 0;
    boiler__holding_readback__reserved_25 AT %IW793 : UINT := 0;
    boiler__holding_readback__reserved_26 AT %IW794 : UINT := 0;
    boiler__holding_readback__reserved_27 AT %IW795 : UINT := 0;
    boiler__holding_readback__reserved_28 AT %IW796 : UINT := 0;
    boiler__holding_readback__blowdown_valve_cmd AT %IW797 : UINT := 0;
    boiler__holding_readback__reserved_30 AT %IW798 : UINT := 0;
    boiler__holding_readback__reserved_31 AT %IW799 : UINT := 0;
    boiler__coil__start AT %QX8.0 : BOOL := FALSE;
    boiler__coil__stop AT %QX8.1 : BOOL := FALSE;
    boiler__coil__reset_trip AT %QX8.2 : BOOL := FALSE;
    boiler__coil__ack_alarm AT %QX8.3 : BOOL := FALSE;
    boiler__coil__emergency_stop AT %QX8.4 : BOOL := FALSE;
    boiler__coil__force_safe AT %QX8.5 : BOOL := FALSE;
    boiler__coil__trip_test AT %QX8.6 : BOOL := FALSE;
    boiler__coil__clear_totalizer AT %QX8.7 : BOOL := FALSE;
    boiler__holding__control_mode AT %QW256 : UINT := 3;
    boiler__holding__command_sequence AT %QW257 : UINT := 0;
    boiler__holding__watchdog_counter AT %QW258 : UINT := 1;
    boiler__holding__reset_key AT %QW259 : UINT := 0;
    boiler__holding__simulation_flags AT %QW260 : UINT := 0;
    boiler__holding__active_controller_id AT %QW261 : UINT := 5;
    boiler__holding__command_lease_time AT %QW262 : UINT := 5;
    boiler__holding__output_rate_limit AT %QW263 : UINT := 1000;
    boiler__holding__reserved AT %QW264 : UINT := 0;
    boiler__holding__primary_setpoint AT %QW265 : UINT := 0;
    boiler__holding__secondary_setpoint AT %QW266 : UINT := 0;
    boiler__holding__manual_output AT %QW267 : UINT := 0;
    boiler__holding__output_high_limit AT %QW268 : UINT := 10000;
    boiler__holding__output_low_limit AT %QW269 : UINT := 0;
    boiler__holding__pid_kp AT %QW275 : UINT := 0;
    boiler__holding__pid_ki AT %QW276 : UINT := 0;
    boiler__holding__pid_kd AT %QW277 : UINT := 0;
    boiler__holding__deadband AT %QW278 : UINT := 0;
    boiler__holding__integral_limit AT %QW279 : UINT := 0;
    boiler__holding__controller_scan_time AT %QW280 : UINT := 200;
    boiler__holding__blowdown_valve_cmd AT %QW285 : UINT := 0;
    steam_valve__input__status_word AT %IW320 : UINT := 0;
    steam_valve__input__alarm_word_1 AT %IW321 : UINT := 0;
    steam_valve__input__alarm_word_2 AT %IW322 : UINT := 0;
    steam_valve__input__trip_word AT %IW323 : UINT := 0;
    steam_valve__input__device_state AT %IW324 : UINT := 0;
    steam_valve__input__first_out_code AT %IW325 : UINT := 0;
    steam_valve__input__overall_quality AT %IW326 : UINT := 0;
    steam_valve__input__register_map_version AT %IW327 : UINT := 0;
    steam_valve__input__firmware_version AT %IW328 : UINT := 0;
    steam_valve__input__command_position AT %IW329 : UINT := 0;
    steam_valve__input__actual_position AT %IW330 : UINT := 0;
    steam_valve__input__upstream_pressure AT %IW331 : UINT := 0;
    steam_valve__input__downstream_pressure AT %IW332 : UINT := 0;
    steam_valve__input__steam_flow AT %IW333 : UINT := 0;
    steam_valve__input__steam_temperature AT %IW334 : UINT := 0;
    steam_valve__input__actuator_speed AT %IW335 : UINT := 0;
    steam_valve__input__position_deviation AT %IW336 : UINT := 0;
    steam_valve__input__fast_close_status AT %IW337 : UINT := 0;
    steam_valve__input__valve_fault_code AT %IW338 : UINT := 0;
    steam_valve__input__reserved_19 AT %IW339 : UINT := 0;
    steam_valve__input__reserved_20 AT %IW340 : UINT := 0;
    steam_valve__input__reserved_21 AT %IW341 : UINT := 0;
    steam_valve__input__reserved_22 AT %IW342 : UINT := 0;
    steam_valve__input__reserved_23 AT %IW343 : UINT := 0;
    steam_valve__input__reserved_24 AT %IW344 : UINT := 0;
    steam_valve__input__reserved_25 AT %IW345 : UINT := 0;
    steam_valve__input__reserved_26 AT %IW346 : UINT := 0;
    steam_valve__input__reserved_27 AT %IW347 : UINT := 0;
    steam_valve__input__reserved_28 AT %IW348 : UINT := 0;
    steam_valve__input__watchdog_echo AT %IW349 : UINT := 0;
    steam_valve__input__scan_time_ms AT %IW350 : UINT := 0;
    steam_valve__input__modbus_request_count AT %IW351 : UINT := 0;
    steam_valve__input__rejected_command_count AT %IW352 : UINT := 0;
    steam_valve__input__exception_count AT %IW353 : UINT := 0;
    steam_valve__input__sim_quality_word AT %IW354 : UINT := 0;
    steam_valve__input__sim_tick_low AT %IW355 : UINT := 0;
    steam_valve__input__comm_loss_seconds AT %IW356 : UINT := 0;
    steam_valve__input__fault_inject_word AT %IW357 : UINT := 0;
    steam_valve__input__snapshot_generation AT %IW358 : UINT := 0;
    steam_valve__input__run_seconds_hi AT %IW359 : UINT := 0;
    steam_valve__input__run_seconds_lo AT %IW360 : UINT := 0;
    steam_valve__input__start_count AT %IW361 : UINT := 0;
    steam_valve__input__trip_count AT %IW362 : UINT := 0;
    steam_valve__input__mass_total_hi AT %IW363 : UINT := 0;
    steam_valve__input__mass_total_lo AT %IW364 : UINT := 0;
    steam_valve__input__energy_total_hi AT %IW365 : UINT := 0;
    steam_valve__input__energy_total_lo AT %IW366 : UINT := 0;
    steam_valve__input__alarm_count AT %IW367 : UINT := 0;
    steam_valve__input__accepted_command_count AT %IW368 : UINT := 0;
    steam_valve__input__reserved_49 AT %IW369 : UINT := 0;
    steam_valve__discrete__ready AT %IX10.0 : BOOL := FALSE;
    steam_valve__discrete__running AT %IX10.1 : BOOL := FALSE;
    steam_valve__discrete__starting AT %IX10.2 : BOOL := FALSE;
    steam_valve__discrete__stopping AT %IX10.3 : BOOL := FALSE;
    steam_valve__discrete__tripped AT %IX10.4 : BOOL := FALSE;
    steam_valve__discrete__alarm_active AT %IX10.5 : BOOL := FALSE;
    steam_valve__discrete__local_mode AT %IX10.6 : BOOL := FALSE;
    steam_valve__discrete__remote_mode AT %IX10.7 : BOOL := FALSE;
    steam_valve__discrete__auto_mode AT %IX11.0 : BOOL := FALSE;
    steam_valve__discrete__manual_mode AT %IX11.1 : BOOL := FALSE;
    steam_valve__discrete__control_watchdog_ok AT %IX11.2 : BOOL := FALSE;
    steam_valve__discrete__sim_bus_ok AT %IX11.3 : BOOL := FALSE;
    steam_valve__discrete__interlocks_ok AT %IX11.4 : BOOL := FALSE;
    steam_valve__discrete__sensor_fault AT %IX11.5 : BOOL := FALSE;
    steam_valve__discrete__actuator_fault AT %IX11.6 : BOOL := FALSE;
    steam_valve__discrete__maintenance_mode AT %IX11.7 : BOOL := FALSE;
    steam_valve__holding_readback__control_mode AT %IW832 : UINT := 0;
    steam_valve__holding_readback__command_sequence AT %IW833 : UINT := 0;
    steam_valve__holding_readback__watchdog_counter AT %IW834 : UINT := 0;
    steam_valve__holding_readback__reset_key AT %IW835 : UINT := 0;
    steam_valve__holding_readback__simulation_flags AT %IW836 : UINT := 0;
    steam_valve__holding_readback__active_controller_id AT %IW837 : UINT := 0;
    steam_valve__holding_readback__command_lease_time AT %IW838 : UINT := 0;
    steam_valve__holding_readback__output_rate_limit AT %IW839 : UINT := 0;
    steam_valve__holding_readback__reserved AT %IW840 : UINT := 0;
    steam_valve__holding_readback__primary_setpoint AT %IW841 : UINT := 0;
    steam_valve__holding_readback__secondary_setpoint AT %IW842 : UINT := 0;
    steam_valve__holding_readback__manual_output AT %IW843 : UINT := 0;
    steam_valve__holding_readback__output_high_limit AT %IW844 : UINT := 0;
    steam_valve__holding_readback__output_low_limit AT %IW845 : UINT := 0;
    steam_valve__holding_readback__reserved_14 AT %IW846 : UINT := 0;
    steam_valve__holding_readback__reserved_15 AT %IW847 : UINT := 0;
    steam_valve__holding_readback__reserved_16 AT %IW848 : UINT := 0;
    steam_valve__holding_readback__reserved_17 AT %IW849 : UINT := 0;
    steam_valve__holding_readback__reserved_18 AT %IW850 : UINT := 0;
    steam_valve__holding_readback__pid_kp AT %IW851 : UINT := 0;
    steam_valve__holding_readback__pid_ki AT %IW852 : UINT := 0;
    steam_valve__holding_readback__pid_kd AT %IW853 : UINT := 0;
    steam_valve__holding_readback__deadband AT %IW854 : UINT := 0;
    steam_valve__holding_readback__integral_limit AT %IW855 : UINT := 0;
    steam_valve__holding_readback__controller_scan_time AT %IW856 : UINT := 0;
    steam_valve__holding_readback__reserved_25 AT %IW857 : UINT := 0;
    steam_valve__holding_readback__reserved_26 AT %IW858 : UINT := 0;
    steam_valve__holding_readback__reserved_27 AT %IW859 : UINT := 0;
    steam_valve__holding_readback__reserved_28 AT %IW860 : UINT := 0;
    steam_valve__holding_readback__open_rate AT %IW861 : UINT := 0;
    steam_valve__holding_readback__close_rate AT %IW862 : UINT := 0;
    steam_valve__holding_readback__reserved_31 AT %IW863 : UINT := 0;
    steam_valve__coil__start AT %QX10.0 : BOOL := FALSE;
    steam_valve__coil__stop AT %QX10.1 : BOOL := FALSE;
    steam_valve__coil__reset_trip AT %QX10.2 : BOOL := FALSE;
    steam_valve__coil__ack_alarm AT %QX10.3 : BOOL := FALSE;
    steam_valve__coil__emergency_stop AT %QX10.4 : BOOL := FALSE;
    steam_valve__coil__force_safe AT %QX10.5 : BOOL := FALSE;
    steam_valve__coil__trip_test AT %QX10.6 : BOOL := FALSE;
    steam_valve__coil__clear_totalizer AT %QX10.7 : BOOL := FALSE;
    steam_valve__holding__control_mode AT %QW320 : UINT := 3;
    steam_valve__holding__command_sequence AT %QW321 : UINT := 0;
    steam_valve__holding__watchdog_counter AT %QW322 : UINT := 1;
    steam_valve__holding__reset_key AT %QW323 : UINT := 0;
    steam_valve__holding__simulation_flags AT %QW324 : UINT := 0;
    steam_valve__holding__active_controller_id AT %QW325 : UINT := 6;
    steam_valve__holding__command_lease_time AT %QW326 : UINT := 5;
    steam_valve__holding__output_rate_limit AT %QW327 : UINT := 1000;
    steam_valve__holding__reserved AT %QW328 : UINT := 0;
    steam_valve__holding__primary_setpoint AT %QW329 : UINT := 0;
    steam_valve__holding__secondary_setpoint AT %QW330 : UINT := 0;
    steam_valve__holding__manual_output AT %QW331 : UINT := 0;
    steam_valve__holding__output_high_limit AT %QW332 : UINT := 10000;
    steam_valve__holding__output_low_limit AT %QW333 : UINT := 0;
    steam_valve__holding__pid_kp AT %QW339 : UINT := 0;
    steam_valve__holding__pid_ki AT %QW340 : UINT := 0;
    steam_valve__holding__pid_kd AT %QW341 : UINT := 0;
    steam_valve__holding__deadband AT %QW342 : UINT := 0;
    steam_valve__holding__integral_limit AT %QW343 : UINT := 0;
    steam_valve__holding__controller_scan_time AT %QW344 : UINT := 200;
    steam_valve__holding__open_rate AT %QW349 : UINT := 10;
    steam_valve__holding__close_rate AT %QW350 : UINT := 10;
    turbine__input__status_word AT %IW384 : UINT := 0;
    turbine__input__alarm_word_1 AT %IW385 : UINT := 0;
    turbine__input__alarm_word_2 AT %IW386 : UINT := 0;
    turbine__input__trip_word AT %IW387 : UINT := 0;
    turbine__input__device_state AT %IW388 : UINT := 0;
    turbine__input__first_out_code AT %IW389 : UINT := 0;
    turbine__input__overall_quality AT %IW390 : UINT := 0;
    turbine__input__register_map_version AT %IW391 : UINT := 0;
    turbine__input__firmware_version AT %IW392 : UINT := 0;
    turbine__input__speed_rpm AT %IW393 : UINT := 0;
    turbine__input__mechanical_power AT %IW394 : UINT := 0;
    turbine__input__steam_flow AT %IW395 : UINT := 0;
    turbine__input__exhaust_flow AT %IW396 : UINT := 0;
    turbine__input__main_steam_pressure AT %IW397 : UINT := 0;
    turbine__input__exhaust_pressure AT %IW398 : UINT := 0;
    turbine__input__vibration AT %IW399 : UINT := 0;
    turbine__input__bearing_temperature AT %IW400 : UINT := 0;
    turbine__input__governor_output AT %IW401 : UINT := 0;
    turbine__input__acceleration AT %IW402 : UINT := 0;
    turbine__input__efficiency AT %IW403 : UINT := 0;
    turbine__input__reserved_20 AT %IW404 : UINT := 0;
    turbine__input__reserved_21 AT %IW405 : UINT := 0;
    turbine__input__reserved_22 AT %IW406 : UINT := 0;
    turbine__input__reserved_23 AT %IW407 : UINT := 0;
    turbine__input__reserved_24 AT %IW408 : UINT := 0;
    turbine__input__reserved_25 AT %IW409 : UINT := 0;
    turbine__input__reserved_26 AT %IW410 : UINT := 0;
    turbine__input__reserved_27 AT %IW411 : UINT := 0;
    turbine__input__reserved_28 AT %IW412 : UINT := 0;
    turbine__input__watchdog_echo AT %IW413 : UINT := 0;
    turbine__input__scan_time_ms AT %IW414 : UINT := 0;
    turbine__input__modbus_request_count AT %IW415 : UINT := 0;
    turbine__input__rejected_command_count AT %IW416 : UINT := 0;
    turbine__input__exception_count AT %IW417 : UINT := 0;
    turbine__input__sim_quality_word AT %IW418 : UINT := 0;
    turbine__input__sim_tick_low AT %IW419 : UINT := 0;
    turbine__input__comm_loss_seconds AT %IW420 : UINT := 0;
    turbine__input__fault_inject_word AT %IW421 : UINT := 0;
    turbine__input__snapshot_generation AT %IW422 : UINT := 0;
    turbine__input__run_seconds_hi AT %IW423 : UINT := 0;
    turbine__input__run_seconds_lo AT %IW424 : UINT := 0;
    turbine__input__start_count AT %IW425 : UINT := 0;
    turbine__input__trip_count AT %IW426 : UINT := 0;
    turbine__input__mass_total_hi AT %IW427 : UINT := 0;
    turbine__input__mass_total_lo AT %IW428 : UINT := 0;
    turbine__input__energy_total_hi AT %IW429 : UINT := 0;
    turbine__input__energy_total_lo AT %IW430 : UINT := 0;
    turbine__input__alarm_count AT %IW431 : UINT := 0;
    turbine__input__accepted_command_count AT %IW432 : UINT := 0;
    turbine__input__reserved_49 AT %IW433 : UINT := 0;
    turbine__discrete__ready AT %IX12.0 : BOOL := FALSE;
    turbine__discrete__running AT %IX12.1 : BOOL := FALSE;
    turbine__discrete__starting AT %IX12.2 : BOOL := FALSE;
    turbine__discrete__stopping AT %IX12.3 : BOOL := FALSE;
    turbine__discrete__tripped AT %IX12.4 : BOOL := FALSE;
    turbine__discrete__alarm_active AT %IX12.5 : BOOL := FALSE;
    turbine__discrete__local_mode AT %IX12.6 : BOOL := FALSE;
    turbine__discrete__remote_mode AT %IX12.7 : BOOL := FALSE;
    turbine__discrete__auto_mode AT %IX13.0 : BOOL := FALSE;
    turbine__discrete__manual_mode AT %IX13.1 : BOOL := FALSE;
    turbine__discrete__control_watchdog_ok AT %IX13.2 : BOOL := FALSE;
    turbine__discrete__sim_bus_ok AT %IX13.3 : BOOL := FALSE;
    turbine__discrete__interlocks_ok AT %IX13.4 : BOOL := FALSE;
    turbine__discrete__sensor_fault AT %IX13.5 : BOOL := FALSE;
    turbine__discrete__actuator_fault AT %IX13.6 : BOOL := FALSE;
    turbine__discrete__maintenance_mode AT %IX13.7 : BOOL := FALSE;
    turbine__holding_readback__control_mode AT %IW896 : UINT := 0;
    turbine__holding_readback__command_sequence AT %IW897 : UINT := 0;
    turbine__holding_readback__watchdog_counter AT %IW898 : UINT := 0;
    turbine__holding_readback__reset_key AT %IW899 : UINT := 0;
    turbine__holding_readback__simulation_flags AT %IW900 : UINT := 0;
    turbine__holding_readback__active_controller_id AT %IW901 : UINT := 0;
    turbine__holding_readback__command_lease_time AT %IW902 : UINT := 0;
    turbine__holding_readback__output_rate_limit AT %IW903 : UINT := 0;
    turbine__holding_readback__reserved AT %IW904 : UINT := 0;
    turbine__holding_readback__primary_setpoint AT %IW905 : UINT := 0;
    turbine__holding_readback__secondary_setpoint AT %IW906 : UINT := 0;
    turbine__holding_readback__manual_output AT %IW907 : UINT := 0;
    turbine__holding_readback__output_high_limit AT %IW908 : UINT := 0;
    turbine__holding_readback__output_low_limit AT %IW909 : UINT := 0;
    turbine__holding_readback__reserved_14 AT %IW910 : UINT := 0;
    turbine__holding_readback__reserved_15 AT %IW911 : UINT := 0;
    turbine__holding_readback__reserved_16 AT %IW912 : UINT := 0;
    turbine__holding_readback__reserved_17 AT %IW913 : UINT := 0;
    turbine__holding_readback__reserved_18 AT %IW914 : UINT := 0;
    turbine__holding_readback__pid_kp AT %IW915 : UINT := 0;
    turbine__holding_readback__pid_ki AT %IW916 : UINT := 0;
    turbine__holding_readback__pid_kd AT %IW917 : UINT := 0;
    turbine__holding_readback__deadband AT %IW918 : UINT := 0;
    turbine__holding_readback__integral_limit AT %IW919 : UINT := 0;
    turbine__holding_readback__controller_scan_time AT %IW920 : UINT := 0;
    turbine__holding_readback__reserved_25 AT %IW921 : UINT := 0;
    turbine__holding_readback__reserved_26 AT %IW922 : UINT := 0;
    turbine__holding_readback__reserved_27 AT %IW923 : UINT := 0;
    turbine__holding_readback__reserved_28 AT %IW924 : UINT := 0;
    turbine__holding_readback__inertia_param AT %IW925 : UINT := 0;
    turbine__holding_readback__damping_param AT %IW926 : UINT := 0;
    turbine__holding_readback__reserved_31 AT %IW927 : UINT := 0;
    turbine__coil__start AT %QX12.0 : BOOL := FALSE;
    turbine__coil__stop AT %QX12.1 : BOOL := FALSE;
    turbine__coil__reset_trip AT %QX12.2 : BOOL := FALSE;
    turbine__coil__ack_alarm AT %QX12.3 : BOOL := FALSE;
    turbine__coil__emergency_stop AT %QX12.4 : BOOL := FALSE;
    turbine__coil__force_safe AT %QX12.5 : BOOL := FALSE;
    turbine__coil__trip_test AT %QX12.6 : BOOL := FALSE;
    turbine__coil__clear_totalizer AT %QX12.7 : BOOL := FALSE;
    turbine__holding__control_mode AT %QW384 : UINT := 3;
    turbine__holding__command_sequence AT %QW385 : UINT := 0;
    turbine__holding__watchdog_counter AT %QW386 : UINT := 1;
    turbine__holding__reset_key AT %QW387 : UINT := 0;
    turbine__holding__simulation_flags AT %QW388 : UINT := 0;
    turbine__holding__active_controller_id AT %QW389 : UINT := 7;
    turbine__holding__command_lease_time AT %QW390 : UINT := 5;
    turbine__holding__output_rate_limit AT %QW391 : UINT := 1000;
    turbine__holding__reserved AT %QW392 : UINT := 0;
    turbine__holding__primary_setpoint AT %QW393 : UINT := 0;
    turbine__holding__secondary_setpoint AT %QW394 : UINT := 0;
    turbine__holding__manual_output AT %QW395 : UINT := 0;
    turbine__holding__output_high_limit AT %QW396 : UINT := 10000;
    turbine__holding__output_low_limit AT %QW397 : UINT := 0;
    turbine__holding__pid_kp AT %QW403 : UINT := 0;
    turbine__holding__pid_ki AT %QW404 : UINT := 0;
    turbine__holding__pid_kd AT %QW405 : UINT := 0;
    turbine__holding__deadband AT %QW406 : UINT := 0;
    turbine__holding__integral_limit AT %QW407 : UINT := 0;
    turbine__holding__controller_scan_time AT %QW408 : UINT := 200;
    turbine__holding__inertia_param AT %QW413 : UINT := 10;
    turbine__holding__damping_param AT %QW414 : UINT := 0;
    generator__input__status_word AT %IW448 : UINT := 0;
    generator__input__alarm_word_1 AT %IW449 : UINT := 0;
    generator__input__alarm_word_2 AT %IW450 : UINT := 0;
    generator__input__trip_word AT %IW451 : UINT := 0;
    generator__input__device_state AT %IW452 : UINT := 0;
    generator__input__first_out_code AT %IW453 : UINT := 0;
    generator__input__overall_quality AT %IW454 : UINT := 0;
    generator__input__register_map_version AT %IW455 : UINT := 0;
    generator__input__firmware_version AT %IW456 : UINT := 0;
    generator__input__electrical_power AT %IW457 : UINT := 0;
    generator__input__load_demand AT %IW458 : UINT := 0;
    generator__input__frequency AT %IW459 : UINT := 0;
    generator__input__voltage AT %IW460 : UINT := 0;
    generator__input__current AT %IW461 : UINT := 0;
    generator__input__power_factor AT %IW462 : UINT := 0;
    generator__input__breaker_status AT %IW463 : UINT := 0;
    generator__input__sync_permissive AT %IW464 : UINT := 0;
    generator__input__phase_angle_diff AT %IW465 : UINT := 0;
    generator__input__electrical_torque AT %IW466 : UINT := 0;
    generator__input__operating_mode AT %IW467 : UINT := 0;
    generator__input__reserved_20 AT %IW468 : UINT := 0;
    generator__input__reserved_21 AT %IW469 : UINT := 0;
    generator__input__reserved_22 AT %IW470 : UINT := 0;
    generator__input__reserved_23 AT %IW471 : UINT := 0;
    generator__input__reserved_24 AT %IW472 : UINT := 0;
    generator__input__reserved_25 AT %IW473 : UINT := 0;
    generator__input__reserved_26 AT %IW474 : UINT := 0;
    generator__input__reserved_27 AT %IW475 : UINT := 0;
    generator__input__reserved_28 AT %IW476 : UINT := 0;
    generator__input__watchdog_echo AT %IW477 : UINT := 0;
    generator__input__scan_time_ms AT %IW478 : UINT := 0;
    generator__input__modbus_request_count AT %IW479 : UINT := 0;
    generator__input__rejected_command_count AT %IW480 : UINT := 0;
    generator__input__exception_count AT %IW481 : UINT := 0;
    generator__input__sim_quality_word AT %IW482 : UINT := 0;
    generator__input__sim_tick_low AT %IW483 : UINT := 0;
    generator__input__comm_loss_seconds AT %IW484 : UINT := 0;
    generator__input__fault_inject_word AT %IW485 : UINT := 0;
    generator__input__snapshot_generation AT %IW486 : UINT := 0;
    generator__input__run_seconds_hi AT %IW487 : UINT := 0;
    generator__input__run_seconds_lo AT %IW488 : UINT := 0;
    generator__input__start_count AT %IW489 : UINT := 0;
    generator__input__trip_count AT %IW490 : UINT := 0;
    generator__input__mass_total_hi AT %IW491 : UINT := 0;
    generator__input__mass_total_lo AT %IW492 : UINT := 0;
    generator__input__energy_total_hi AT %IW493 : UINT := 0;
    generator__input__energy_total_lo AT %IW494 : UINT := 0;
    generator__input__alarm_count AT %IW495 : UINT := 0;
    generator__input__accepted_command_count AT %IW496 : UINT := 0;
    generator__input__reserved_49 AT %IW497 : UINT := 0;
    generator__discrete__ready AT %IX14.0 : BOOL := FALSE;
    generator__discrete__running AT %IX14.1 : BOOL := FALSE;
    generator__discrete__starting AT %IX14.2 : BOOL := FALSE;
    generator__discrete__stopping AT %IX14.3 : BOOL := FALSE;
    generator__discrete__tripped AT %IX14.4 : BOOL := FALSE;
    generator__discrete__alarm_active AT %IX14.5 : BOOL := FALSE;
    generator__discrete__local_mode AT %IX14.6 : BOOL := FALSE;
    generator__discrete__remote_mode AT %IX14.7 : BOOL := FALSE;
    generator__discrete__auto_mode AT %IX15.0 : BOOL := FALSE;
    generator__discrete__manual_mode AT %IX15.1 : BOOL := FALSE;
    generator__discrete__control_watchdog_ok AT %IX15.2 : BOOL := FALSE;
    generator__discrete__sim_bus_ok AT %IX15.3 : BOOL := FALSE;
    generator__discrete__interlocks_ok AT %IX15.4 : BOOL := FALSE;
    generator__discrete__sensor_fault AT %IX15.5 : BOOL := FALSE;
    generator__discrete__actuator_fault AT %IX15.6 : BOOL := FALSE;
    generator__discrete__maintenance_mode AT %IX15.7 : BOOL := FALSE;
    generator__holding_readback__control_mode AT %IW960 : UINT := 0;
    generator__holding_readback__command_sequence AT %IW961 : UINT := 0;
    generator__holding_readback__watchdog_counter AT %IW962 : UINT := 0;
    generator__holding_readback__reset_key AT %IW963 : UINT := 0;
    generator__holding_readback__simulation_flags AT %IW964 : UINT := 0;
    generator__holding_readback__active_controller_id AT %IW965 : UINT := 0;
    generator__holding_readback__command_lease_time AT %IW966 : UINT := 0;
    generator__holding_readback__output_rate_limit AT %IW967 : UINT := 0;
    generator__holding_readback__reserved AT %IW968 : UINT := 0;
    generator__holding_readback__primary_setpoint AT %IW969 : UINT := 0;
    generator__holding_readback__secondary_setpoint AT %IW970 : UINT := 0;
    generator__holding_readback__manual_output AT %IW971 : UINT := 0;
    generator__holding_readback__output_high_limit AT %IW972 : UINT := 0;
    generator__holding_readback__output_low_limit AT %IW973 : UINT := 0;
    generator__holding_readback__reserved_14 AT %IW974 : UINT := 0;
    generator__holding_readback__reserved_15 AT %IW975 : UINT := 0;
    generator__holding_readback__reserved_16 AT %IW976 : UINT := 0;
    generator__holding_readback__reserved_17 AT %IW977 : UINT := 0;
    generator__holding_readback__reserved_18 AT %IW978 : UINT := 0;
    generator__holding_readback__pid_kp AT %IW979 : UINT := 0;
    generator__holding_readback__pid_ki AT %IW980 : UINT := 0;
    generator__holding_readback__pid_kd AT %IW981 : UINT := 0;
    generator__holding_readback__deadband AT %IW982 : UINT := 0;
    generator__holding_readback__integral_limit AT %IW983 : UINT := 0;
    generator__holding_readback__controller_scan_time AT %IW984 : UINT := 0;
    generator__holding_readback__reserved_25 AT %IW985 : UINT := 0;
    generator__holding_readback__reserved_26 AT %IW986 : UINT := 0;
    generator__holding_readback__reserved_27 AT %IW987 : UINT := 0;
    generator__holding_readback__reserved_28 AT %IW988 : UINT := 0;
    generator__holding_readback__operating_mode AT %IW989 : UINT := 0;
    generator__holding_readback__load_rate_limit AT %IW990 : UINT := 0;
    generator__holding_readback__reserved_31 AT %IW991 : UINT := 0;
    generator__coil__start AT %QX14.0 : BOOL := FALSE;
    generator__coil__stop AT %QX14.1 : BOOL := FALSE;
    generator__coil__reset_trip AT %QX14.2 : BOOL := FALSE;
    generator__coil__ack_alarm AT %QX14.3 : BOOL := FALSE;
    generator__coil__emergency_stop AT %QX14.4 : BOOL := FALSE;
    generator__coil__force_safe AT %QX14.5 : BOOL := FALSE;
    generator__coil__trip_test AT %QX14.6 : BOOL := FALSE;
    generator__coil__clear_totalizer AT %QX14.7 : BOOL := FALSE;
    generator__coil__breaker_close AT %QX15.1 : BOOL := FALSE;
    generator__coil__breaker_open AT %QX15.2 : BOOL := FALSE;
    generator__holding__control_mode AT %QW448 : UINT := 3;
    generator__holding__command_sequence AT %QW449 : UINT := 0;
    generator__holding__watchdog_counter AT %QW450 : UINT := 1;
    generator__holding__reset_key AT %QW451 : UINT := 0;
    generator__holding__simulation_flags AT %QW452 : UINT := 0;
    generator__holding__active_controller_id AT %QW453 : UINT := 8;
    generator__holding__command_lease_time AT %QW454 : UINT := 5;
    generator__holding__output_rate_limit AT %QW455 : UINT := 1000;
    generator__holding__reserved AT %QW456 : UINT := 0;
    generator__holding__primary_setpoint AT %QW457 : UINT := 0;
    generator__holding__secondary_setpoint AT %QW458 : UINT := 0;
    generator__holding__manual_output AT %QW459 : UINT := 0;
    generator__holding__output_high_limit AT %QW460 : UINT := 10000;
    generator__holding__output_low_limit AT %QW461 : UINT := 0;
    generator__holding__pid_kp AT %QW467 : UINT := 0;
    generator__holding__pid_ki AT %QW468 : UINT := 0;
    generator__holding__pid_kd AT %QW469 : UINT := 0;
    generator__holding__deadband AT %QW470 : UINT := 0;
    generator__holding__integral_limit AT %QW471 : UINT := 0;
    generator__holding__controller_scan_time AT %QW472 : UINT := 200;
    generator__holding__operating_mode AT %QW477 : UINT := 0;
    generator__holding__load_rate_limit AT %QW478 : UINT := 10;
  END_VAR

  (* 200 ms non-zero watchdog for every device. *)
  i_watchdog_tick := FALSE;
  i_watchdog_scan_count := i_watchdog_scan_count + 1;
  IF i_watchdog_scan_count >= 10 THEN
    i_watchdog_scan_count := 0;
    i_watchdog_tick := TRUE;
    IF condenser__holding__watchdog_counter >= 65535 THEN
      condenser__holding__watchdog_counter := 1;
    ELSE
      condenser__holding__watchdog_counter := condenser__holding__watchdog_counter + 1;
    END_IF;
    IF condensate_pump__holding__watchdog_counter >= 65535 THEN
      condensate_pump__holding__watchdog_counter := 1;
    ELSE
      condensate_pump__holding__watchdog_counter := condensate_pump__holding__watchdog_counter + 1;
    END_IF;
    IF feedwater_tank__holding__watchdog_counter >= 65535 THEN
      feedwater_tank__holding__watchdog_counter := 1;
    ELSE
      feedwater_tank__holding__watchdog_counter := feedwater_tank__holding__watchdog_counter + 1;
    END_IF;
    IF feedwater_pump__holding__watchdog_counter >= 65535 THEN
      feedwater_pump__holding__watchdog_counter := 1;
    ELSE
      feedwater_pump__holding__watchdog_counter := feedwater_pump__holding__watchdog_counter + 1;
    END_IF;
    IF boiler__holding__watchdog_counter >= 65535 THEN
      boiler__holding__watchdog_counter := 1;
    ELSE
      boiler__holding__watchdog_counter := boiler__holding__watchdog_counter + 1;
    END_IF;
    IF steam_valve__holding__watchdog_counter >= 65535 THEN
      steam_valve__holding__watchdog_counter := 1;
    ELSE
      steam_valve__holding__watchdog_counter := steam_valve__holding__watchdog_counter + 1;
    END_IF;
    IF turbine__holding__watchdog_counter >= 65535 THEN
      turbine__holding__watchdog_counter := 1;
    ELSE
      turbine__holding__watchdog_counter := turbine__holding__watchdog_counter + 1;
    END_IF;
    IF generator__holding__watchdog_counter >= 65535 THEN
      generator__holding__watchdog_counter := 1;
    ELSE
      generator__holding__watchdog_counter := generator__holding__watchdog_counter + 1;
    END_IF;
  END_IF;

  (* Echo may lag the current counter because FC4 polls every 250 ms.
     Progress or equality proves the link; an unchanged mismatch for
     15 watchdog ticks (3 s) is a communication failure. *)
  IF i_watchdog_tick THEN
    IF (condenser__input__watchdog_echo = condenser__holding__watchdog_counter) OR (condenser__input__watchdog_echo <> i_condenser_last_echo) THEN
      i_condenser_last_echo := condenser__input__watchdog_echo;
      i_condenser_echo_stale_ticks := 0;
    ELSE
      IF i_condenser_echo_stale_ticks < 65535 THEN
        i_condenser_echo_stale_ticks := i_condenser_echo_stale_ticks + 1;
      END_IF;
    END_IF;
    i_condenser_comm_lost := i_condenser_echo_stale_ticks >= 15;
    IF (condensate_pump__input__watchdog_echo = condensate_pump__holding__watchdog_counter) OR (condensate_pump__input__watchdog_echo <> i_condensate_pump_last_echo) THEN
      i_condensate_pump_last_echo := condensate_pump__input__watchdog_echo;
      i_condensate_pump_echo_stale_ticks := 0;
    ELSE
      IF i_condensate_pump_echo_stale_ticks < 65535 THEN
        i_condensate_pump_echo_stale_ticks := i_condensate_pump_echo_stale_ticks + 1;
      END_IF;
    END_IF;
    i_condensate_pump_comm_lost := i_condensate_pump_echo_stale_ticks >= 15;
    IF (feedwater_tank__input__watchdog_echo = feedwater_tank__holding__watchdog_counter) OR (feedwater_tank__input__watchdog_echo <> i_feedwater_tank_last_echo) THEN
      i_feedwater_tank_last_echo := feedwater_tank__input__watchdog_echo;
      i_feedwater_tank_echo_stale_ticks := 0;
    ELSE
      IF i_feedwater_tank_echo_stale_ticks < 65535 THEN
        i_feedwater_tank_echo_stale_ticks := i_feedwater_tank_echo_stale_ticks + 1;
      END_IF;
    END_IF;
    i_feedwater_tank_comm_lost := i_feedwater_tank_echo_stale_ticks >= 15;
    IF (feedwater_pump__input__watchdog_echo = feedwater_pump__holding__watchdog_counter) OR (feedwater_pump__input__watchdog_echo <> i_feedwater_pump_last_echo) THEN
      i_feedwater_pump_last_echo := feedwater_pump__input__watchdog_echo;
      i_feedwater_pump_echo_stale_ticks := 0;
    ELSE
      IF i_feedwater_pump_echo_stale_ticks < 65535 THEN
        i_feedwater_pump_echo_stale_ticks := i_feedwater_pump_echo_stale_ticks + 1;
      END_IF;
    END_IF;
    i_feedwater_pump_comm_lost := i_feedwater_pump_echo_stale_ticks >= 15;
    IF (boiler__input__watchdog_echo = boiler__holding__watchdog_counter) OR (boiler__input__watchdog_echo <> i_boiler_last_echo) THEN
      i_boiler_last_echo := boiler__input__watchdog_echo;
      i_boiler_echo_stale_ticks := 0;
    ELSE
      IF i_boiler_echo_stale_ticks < 65535 THEN
        i_boiler_echo_stale_ticks := i_boiler_echo_stale_ticks + 1;
      END_IF;
    END_IF;
    i_boiler_comm_lost := i_boiler_echo_stale_ticks >= 15;
    IF (steam_valve__input__watchdog_echo = steam_valve__holding__watchdog_counter) OR (steam_valve__input__watchdog_echo <> i_steam_valve_last_echo) THEN
      i_steam_valve_last_echo := steam_valve__input__watchdog_echo;
      i_steam_valve_echo_stale_ticks := 0;
    ELSE
      IF i_steam_valve_echo_stale_ticks < 65535 THEN
        i_steam_valve_echo_stale_ticks := i_steam_valve_echo_stale_ticks + 1;
      END_IF;
    END_IF;
    i_steam_valve_comm_lost := i_steam_valve_echo_stale_ticks >= 15;
    IF (turbine__input__watchdog_echo = turbine__holding__watchdog_counter) OR (turbine__input__watchdog_echo <> i_turbine_last_echo) THEN
      i_turbine_last_echo := turbine__input__watchdog_echo;
      i_turbine_echo_stale_ticks := 0;
    ELSE
      IF i_turbine_echo_stale_ticks < 65535 THEN
        i_turbine_echo_stale_ticks := i_turbine_echo_stale_ticks + 1;
      END_IF;
    END_IF;
    i_turbine_comm_lost := i_turbine_echo_stale_ticks >= 15;
    IF (generator__input__watchdog_echo = generator__holding__watchdog_counter) OR (generator__input__watchdog_echo <> i_generator_last_echo) THEN
      i_generator_last_echo := generator__input__watchdog_echo;
      i_generator_echo_stale_ticks := 0;
    ELSE
      IF i_generator_echo_stale_ticks < 65535 THEN
        i_generator_echo_stale_ticks := i_generator_echo_stale_ticks + 1;
      END_IF;
    END_IF;
    i_generator_comm_lost := i_generator_echo_stale_ticks >= 15;
  END_IF;

  (* Communication fail-safe matrix from docs/plc-integration.md. *)
  IF i_condenser_comm_lost THEN
    condenser__holding__control_mode := 1;
  END_IF;
  IF i_condensate_pump_comm_lost THEN
    condensate_pump__holding__control_mode := 1;
  END_IF;
  IF i_boiler_comm_lost THEN
    boiler__holding__manual_output := 0;
  END_IF;
  IF i_turbine_comm_lost THEN
    turbine__holding__manual_output := 0;
  END_IF;
  IF i_steam_valve_comm_lost THEN
    steam_valve__holding__manual_output := 0;
  END_IF;
  (* feedwater_pump/feedwater_tank/generator intentionally HOLD_LAST. *)

  (* Pulse outputs are stretched to about 160 ms then cleared.
     EMERGENCY_STOP and FORCE_SAFE are deliberately not included. *)
  IF condenser__coil__start AND NOT i_condenser_start_active THEN
    i_condenser_start_active := TRUE;
    i_condenser_start_scans := 0;
  END_IF;
  IF i_condenser_start_active THEN
    i_condenser_start_scans := i_condenser_start_scans + 1;
    IF i_condenser_start_scans >= 8 THEN
      condenser__coil__start := FALSE;
      i_condenser_start_active := FALSE;
      i_condenser_start_scans := 0;
    END_IF;
  END_IF;
  IF condenser__coil__stop AND NOT i_condenser_stop_active THEN
    i_condenser_stop_active := TRUE;
    i_condenser_stop_scans := 0;
  END_IF;
  IF i_condenser_stop_active THEN
    i_condenser_stop_scans := i_condenser_stop_scans + 1;
    IF i_condenser_stop_scans >= 8 THEN
      condenser__coil__stop := FALSE;
      i_condenser_stop_active := FALSE;
      i_condenser_stop_scans := 0;
    END_IF;
  END_IF;
  IF condenser__coil__reset_trip AND NOT i_condenser_reset_trip_active THEN
    i_condenser_reset_trip_active := TRUE;
    i_condenser_reset_trip_scans := 0;
    IF condenser__holding__command_sequence >= 65535 THEN
      condenser__holding__command_sequence := 1;
    ELSE
      condenser__holding__command_sequence := condenser__holding__command_sequence + 1;
    END_IF;
    condenser__holding__reset_key := 42330;
  END_IF;
  IF i_condenser_reset_trip_active THEN
    i_condenser_reset_trip_scans := i_condenser_reset_trip_scans + 1;
    IF i_condenser_reset_trip_scans >= 8 THEN
      condenser__coil__reset_trip := FALSE;
      i_condenser_reset_trip_active := FALSE;
      i_condenser_reset_trip_scans := 0;
      condenser__holding__reset_key := 0;
    END_IF;
  END_IF;
  IF condenser__coil__ack_alarm AND NOT i_condenser_ack_alarm_active THEN
    i_condenser_ack_alarm_active := TRUE;
    i_condenser_ack_alarm_scans := 0;
  END_IF;
  IF i_condenser_ack_alarm_active THEN
    i_condenser_ack_alarm_scans := i_condenser_ack_alarm_scans + 1;
    IF i_condenser_ack_alarm_scans >= 8 THEN
      condenser__coil__ack_alarm := FALSE;
      i_condenser_ack_alarm_active := FALSE;
      i_condenser_ack_alarm_scans := 0;
    END_IF;
  END_IF;
  IF condenser__coil__trip_test AND NOT i_condenser_trip_test_active THEN
    i_condenser_trip_test_active := TRUE;
    i_condenser_trip_test_scans := 0;
  END_IF;
  IF i_condenser_trip_test_active THEN
    i_condenser_trip_test_scans := i_condenser_trip_test_scans + 1;
    IF i_condenser_trip_test_scans >= 8 THEN
      condenser__coil__trip_test := FALSE;
      i_condenser_trip_test_active := FALSE;
      i_condenser_trip_test_scans := 0;
    END_IF;
  END_IF;
  IF condenser__coil__clear_totalizer AND NOT i_condenser_clear_totalizer_active THEN
    i_condenser_clear_totalizer_active := TRUE;
    i_condenser_clear_totalizer_scans := 0;
  END_IF;
  IF i_condenser_clear_totalizer_active THEN
    i_condenser_clear_totalizer_scans := i_condenser_clear_totalizer_scans + 1;
    IF i_condenser_clear_totalizer_scans >= 8 THEN
      condenser__coil__clear_totalizer := FALSE;
      i_condenser_clear_totalizer_active := FALSE;
      i_condenser_clear_totalizer_scans := 0;
    END_IF;
  END_IF;
  IF condensate_pump__coil__start AND NOT i_condensate_pump_start_active THEN
    i_condensate_pump_start_active := TRUE;
    i_condensate_pump_start_scans := 0;
  END_IF;
  IF i_condensate_pump_start_active THEN
    i_condensate_pump_start_scans := i_condensate_pump_start_scans + 1;
    IF i_condensate_pump_start_scans >= 8 THEN
      condensate_pump__coil__start := FALSE;
      i_condensate_pump_start_active := FALSE;
      i_condensate_pump_start_scans := 0;
    END_IF;
  END_IF;
  IF condensate_pump__coil__stop AND NOT i_condensate_pump_stop_active THEN
    i_condensate_pump_stop_active := TRUE;
    i_condensate_pump_stop_scans := 0;
  END_IF;
  IF i_condensate_pump_stop_active THEN
    i_condensate_pump_stop_scans := i_condensate_pump_stop_scans + 1;
    IF i_condensate_pump_stop_scans >= 8 THEN
      condensate_pump__coil__stop := FALSE;
      i_condensate_pump_stop_active := FALSE;
      i_condensate_pump_stop_scans := 0;
    END_IF;
  END_IF;
  IF condensate_pump__coil__reset_trip AND NOT i_condensate_pump_reset_trip_active THEN
    i_condensate_pump_reset_trip_active := TRUE;
    i_condensate_pump_reset_trip_scans := 0;
    IF condensate_pump__holding__command_sequence >= 65535 THEN
      condensate_pump__holding__command_sequence := 1;
    ELSE
      condensate_pump__holding__command_sequence := condensate_pump__holding__command_sequence + 1;
    END_IF;
    condensate_pump__holding__reset_key := 42330;
  END_IF;
  IF i_condensate_pump_reset_trip_active THEN
    i_condensate_pump_reset_trip_scans := i_condensate_pump_reset_trip_scans + 1;
    IF i_condensate_pump_reset_trip_scans >= 8 THEN
      condensate_pump__coil__reset_trip := FALSE;
      i_condensate_pump_reset_trip_active := FALSE;
      i_condensate_pump_reset_trip_scans := 0;
      condensate_pump__holding__reset_key := 0;
    END_IF;
  END_IF;
  IF condensate_pump__coil__ack_alarm AND NOT i_condensate_pump_ack_alarm_active THEN
    i_condensate_pump_ack_alarm_active := TRUE;
    i_condensate_pump_ack_alarm_scans := 0;
  END_IF;
  IF i_condensate_pump_ack_alarm_active THEN
    i_condensate_pump_ack_alarm_scans := i_condensate_pump_ack_alarm_scans + 1;
    IF i_condensate_pump_ack_alarm_scans >= 8 THEN
      condensate_pump__coil__ack_alarm := FALSE;
      i_condensate_pump_ack_alarm_active := FALSE;
      i_condensate_pump_ack_alarm_scans := 0;
    END_IF;
  END_IF;
  IF condensate_pump__coil__trip_test AND NOT i_condensate_pump_trip_test_active THEN
    i_condensate_pump_trip_test_active := TRUE;
    i_condensate_pump_trip_test_scans := 0;
  END_IF;
  IF i_condensate_pump_trip_test_active THEN
    i_condensate_pump_trip_test_scans := i_condensate_pump_trip_test_scans + 1;
    IF i_condensate_pump_trip_test_scans >= 8 THEN
      condensate_pump__coil__trip_test := FALSE;
      i_condensate_pump_trip_test_active := FALSE;
      i_condensate_pump_trip_test_scans := 0;
    END_IF;
  END_IF;
  IF condensate_pump__coil__clear_totalizer AND NOT i_condensate_pump_clear_totalizer_active THEN
    i_condensate_pump_clear_totalizer_active := TRUE;
    i_condensate_pump_clear_totalizer_scans := 0;
  END_IF;
  IF i_condensate_pump_clear_totalizer_active THEN
    i_condensate_pump_clear_totalizer_scans := i_condensate_pump_clear_totalizer_scans + 1;
    IF i_condensate_pump_clear_totalizer_scans >= 8 THEN
      condensate_pump__coil__clear_totalizer := FALSE;
      i_condensate_pump_clear_totalizer_active := FALSE;
      i_condensate_pump_clear_totalizer_scans := 0;
    END_IF;
  END_IF;
  IF feedwater_tank__coil__start AND NOT i_feedwater_tank_start_active THEN
    i_feedwater_tank_start_active := TRUE;
    i_feedwater_tank_start_scans := 0;
  END_IF;
  IF i_feedwater_tank_start_active THEN
    i_feedwater_tank_start_scans := i_feedwater_tank_start_scans + 1;
    IF i_feedwater_tank_start_scans >= 8 THEN
      feedwater_tank__coil__start := FALSE;
      i_feedwater_tank_start_active := FALSE;
      i_feedwater_tank_start_scans := 0;
    END_IF;
  END_IF;
  IF feedwater_tank__coil__stop AND NOT i_feedwater_tank_stop_active THEN
    i_feedwater_tank_stop_active := TRUE;
    i_feedwater_tank_stop_scans := 0;
  END_IF;
  IF i_feedwater_tank_stop_active THEN
    i_feedwater_tank_stop_scans := i_feedwater_tank_stop_scans + 1;
    IF i_feedwater_tank_stop_scans >= 8 THEN
      feedwater_tank__coil__stop := FALSE;
      i_feedwater_tank_stop_active := FALSE;
      i_feedwater_tank_stop_scans := 0;
    END_IF;
  END_IF;
  IF feedwater_tank__coil__reset_trip AND NOT i_feedwater_tank_reset_trip_active THEN
    i_feedwater_tank_reset_trip_active := TRUE;
    i_feedwater_tank_reset_trip_scans := 0;
    IF feedwater_tank__holding__command_sequence >= 65535 THEN
      feedwater_tank__holding__command_sequence := 1;
    ELSE
      feedwater_tank__holding__command_sequence := feedwater_tank__holding__command_sequence + 1;
    END_IF;
    feedwater_tank__holding__reset_key := 42330;
  END_IF;
  IF i_feedwater_tank_reset_trip_active THEN
    i_feedwater_tank_reset_trip_scans := i_feedwater_tank_reset_trip_scans + 1;
    IF i_feedwater_tank_reset_trip_scans >= 8 THEN
      feedwater_tank__coil__reset_trip := FALSE;
      i_feedwater_tank_reset_trip_active := FALSE;
      i_feedwater_tank_reset_trip_scans := 0;
      feedwater_tank__holding__reset_key := 0;
    END_IF;
  END_IF;
  IF feedwater_tank__coil__ack_alarm AND NOT i_feedwater_tank_ack_alarm_active THEN
    i_feedwater_tank_ack_alarm_active := TRUE;
    i_feedwater_tank_ack_alarm_scans := 0;
  END_IF;
  IF i_feedwater_tank_ack_alarm_active THEN
    i_feedwater_tank_ack_alarm_scans := i_feedwater_tank_ack_alarm_scans + 1;
    IF i_feedwater_tank_ack_alarm_scans >= 8 THEN
      feedwater_tank__coil__ack_alarm := FALSE;
      i_feedwater_tank_ack_alarm_active := FALSE;
      i_feedwater_tank_ack_alarm_scans := 0;
    END_IF;
  END_IF;
  IF feedwater_tank__coil__trip_test AND NOT i_feedwater_tank_trip_test_active THEN
    i_feedwater_tank_trip_test_active := TRUE;
    i_feedwater_tank_trip_test_scans := 0;
  END_IF;
  IF i_feedwater_tank_trip_test_active THEN
    i_feedwater_tank_trip_test_scans := i_feedwater_tank_trip_test_scans + 1;
    IF i_feedwater_tank_trip_test_scans >= 8 THEN
      feedwater_tank__coil__trip_test := FALSE;
      i_feedwater_tank_trip_test_active := FALSE;
      i_feedwater_tank_trip_test_scans := 0;
    END_IF;
  END_IF;
  IF feedwater_tank__coil__clear_totalizer AND NOT i_feedwater_tank_clear_totalizer_active THEN
    i_feedwater_tank_clear_totalizer_active := TRUE;
    i_feedwater_tank_clear_totalizer_scans := 0;
  END_IF;
  IF i_feedwater_tank_clear_totalizer_active THEN
    i_feedwater_tank_clear_totalizer_scans := i_feedwater_tank_clear_totalizer_scans + 1;
    IF i_feedwater_tank_clear_totalizer_scans >= 8 THEN
      feedwater_tank__coil__clear_totalizer := FALSE;
      i_feedwater_tank_clear_totalizer_active := FALSE;
      i_feedwater_tank_clear_totalizer_scans := 0;
    END_IF;
  END_IF;
  IF feedwater_pump__coil__start AND NOT i_feedwater_pump_start_active THEN
    i_feedwater_pump_start_active := TRUE;
    i_feedwater_pump_start_scans := 0;
  END_IF;
  IF i_feedwater_pump_start_active THEN
    i_feedwater_pump_start_scans := i_feedwater_pump_start_scans + 1;
    IF i_feedwater_pump_start_scans >= 8 THEN
      feedwater_pump__coil__start := FALSE;
      i_feedwater_pump_start_active := FALSE;
      i_feedwater_pump_start_scans := 0;
    END_IF;
  END_IF;
  IF feedwater_pump__coil__stop AND NOT i_feedwater_pump_stop_active THEN
    i_feedwater_pump_stop_active := TRUE;
    i_feedwater_pump_stop_scans := 0;
  END_IF;
  IF i_feedwater_pump_stop_active THEN
    i_feedwater_pump_stop_scans := i_feedwater_pump_stop_scans + 1;
    IF i_feedwater_pump_stop_scans >= 8 THEN
      feedwater_pump__coil__stop := FALSE;
      i_feedwater_pump_stop_active := FALSE;
      i_feedwater_pump_stop_scans := 0;
    END_IF;
  END_IF;
  IF feedwater_pump__coil__reset_trip AND NOT i_feedwater_pump_reset_trip_active THEN
    i_feedwater_pump_reset_trip_active := TRUE;
    i_feedwater_pump_reset_trip_scans := 0;
    IF feedwater_pump__holding__command_sequence >= 65535 THEN
      feedwater_pump__holding__command_sequence := 1;
    ELSE
      feedwater_pump__holding__command_sequence := feedwater_pump__holding__command_sequence + 1;
    END_IF;
    feedwater_pump__holding__reset_key := 42330;
  END_IF;
  IF i_feedwater_pump_reset_trip_active THEN
    i_feedwater_pump_reset_trip_scans := i_feedwater_pump_reset_trip_scans + 1;
    IF i_feedwater_pump_reset_trip_scans >= 8 THEN
      feedwater_pump__coil__reset_trip := FALSE;
      i_feedwater_pump_reset_trip_active := FALSE;
      i_feedwater_pump_reset_trip_scans := 0;
      feedwater_pump__holding__reset_key := 0;
    END_IF;
  END_IF;
  IF feedwater_pump__coil__ack_alarm AND NOT i_feedwater_pump_ack_alarm_active THEN
    i_feedwater_pump_ack_alarm_active := TRUE;
    i_feedwater_pump_ack_alarm_scans := 0;
  END_IF;
  IF i_feedwater_pump_ack_alarm_active THEN
    i_feedwater_pump_ack_alarm_scans := i_feedwater_pump_ack_alarm_scans + 1;
    IF i_feedwater_pump_ack_alarm_scans >= 8 THEN
      feedwater_pump__coil__ack_alarm := FALSE;
      i_feedwater_pump_ack_alarm_active := FALSE;
      i_feedwater_pump_ack_alarm_scans := 0;
    END_IF;
  END_IF;
  IF feedwater_pump__coil__trip_test AND NOT i_feedwater_pump_trip_test_active THEN
    i_feedwater_pump_trip_test_active := TRUE;
    i_feedwater_pump_trip_test_scans := 0;
  END_IF;
  IF i_feedwater_pump_trip_test_active THEN
    i_feedwater_pump_trip_test_scans := i_feedwater_pump_trip_test_scans + 1;
    IF i_feedwater_pump_trip_test_scans >= 8 THEN
      feedwater_pump__coil__trip_test := FALSE;
      i_feedwater_pump_trip_test_active := FALSE;
      i_feedwater_pump_trip_test_scans := 0;
    END_IF;
  END_IF;
  IF feedwater_pump__coil__clear_totalizer AND NOT i_feedwater_pump_clear_totalizer_active THEN
    i_feedwater_pump_clear_totalizer_active := TRUE;
    i_feedwater_pump_clear_totalizer_scans := 0;
  END_IF;
  IF i_feedwater_pump_clear_totalizer_active THEN
    i_feedwater_pump_clear_totalizer_scans := i_feedwater_pump_clear_totalizer_scans + 1;
    IF i_feedwater_pump_clear_totalizer_scans >= 8 THEN
      feedwater_pump__coil__clear_totalizer := FALSE;
      i_feedwater_pump_clear_totalizer_active := FALSE;
      i_feedwater_pump_clear_totalizer_scans := 0;
    END_IF;
  END_IF;
  IF boiler__coil__start AND NOT i_boiler_start_active THEN
    i_boiler_start_active := TRUE;
    i_boiler_start_scans := 0;
  END_IF;
  IF i_boiler_start_active THEN
    i_boiler_start_scans := i_boiler_start_scans + 1;
    IF i_boiler_start_scans >= 8 THEN
      boiler__coil__start := FALSE;
      i_boiler_start_active := FALSE;
      i_boiler_start_scans := 0;
    END_IF;
  END_IF;
  IF boiler__coil__stop AND NOT i_boiler_stop_active THEN
    i_boiler_stop_active := TRUE;
    i_boiler_stop_scans := 0;
  END_IF;
  IF i_boiler_stop_active THEN
    i_boiler_stop_scans := i_boiler_stop_scans + 1;
    IF i_boiler_stop_scans >= 8 THEN
      boiler__coil__stop := FALSE;
      i_boiler_stop_active := FALSE;
      i_boiler_stop_scans := 0;
    END_IF;
  END_IF;
  IF boiler__coil__reset_trip AND NOT i_boiler_reset_trip_active THEN
    i_boiler_reset_trip_active := TRUE;
    i_boiler_reset_trip_scans := 0;
    IF boiler__holding__command_sequence >= 65535 THEN
      boiler__holding__command_sequence := 1;
    ELSE
      boiler__holding__command_sequence := boiler__holding__command_sequence + 1;
    END_IF;
    boiler__holding__reset_key := 42330;
  END_IF;
  IF i_boiler_reset_trip_active THEN
    i_boiler_reset_trip_scans := i_boiler_reset_trip_scans + 1;
    IF i_boiler_reset_trip_scans >= 8 THEN
      boiler__coil__reset_trip := FALSE;
      i_boiler_reset_trip_active := FALSE;
      i_boiler_reset_trip_scans := 0;
      boiler__holding__reset_key := 0;
    END_IF;
  END_IF;
  IF boiler__coil__ack_alarm AND NOT i_boiler_ack_alarm_active THEN
    i_boiler_ack_alarm_active := TRUE;
    i_boiler_ack_alarm_scans := 0;
  END_IF;
  IF i_boiler_ack_alarm_active THEN
    i_boiler_ack_alarm_scans := i_boiler_ack_alarm_scans + 1;
    IF i_boiler_ack_alarm_scans >= 8 THEN
      boiler__coil__ack_alarm := FALSE;
      i_boiler_ack_alarm_active := FALSE;
      i_boiler_ack_alarm_scans := 0;
    END_IF;
  END_IF;
  IF boiler__coil__trip_test AND NOT i_boiler_trip_test_active THEN
    i_boiler_trip_test_active := TRUE;
    i_boiler_trip_test_scans := 0;
  END_IF;
  IF i_boiler_trip_test_active THEN
    i_boiler_trip_test_scans := i_boiler_trip_test_scans + 1;
    IF i_boiler_trip_test_scans >= 8 THEN
      boiler__coil__trip_test := FALSE;
      i_boiler_trip_test_active := FALSE;
      i_boiler_trip_test_scans := 0;
    END_IF;
  END_IF;
  IF boiler__coil__clear_totalizer AND NOT i_boiler_clear_totalizer_active THEN
    i_boiler_clear_totalizer_active := TRUE;
    i_boiler_clear_totalizer_scans := 0;
  END_IF;
  IF i_boiler_clear_totalizer_active THEN
    i_boiler_clear_totalizer_scans := i_boiler_clear_totalizer_scans + 1;
    IF i_boiler_clear_totalizer_scans >= 8 THEN
      boiler__coil__clear_totalizer := FALSE;
      i_boiler_clear_totalizer_active := FALSE;
      i_boiler_clear_totalizer_scans := 0;
    END_IF;
  END_IF;
  IF steam_valve__coil__start AND NOT i_steam_valve_start_active THEN
    i_steam_valve_start_active := TRUE;
    i_steam_valve_start_scans := 0;
  END_IF;
  IF i_steam_valve_start_active THEN
    i_steam_valve_start_scans := i_steam_valve_start_scans + 1;
    IF i_steam_valve_start_scans >= 8 THEN
      steam_valve__coil__start := FALSE;
      i_steam_valve_start_active := FALSE;
      i_steam_valve_start_scans := 0;
    END_IF;
  END_IF;
  IF steam_valve__coil__stop AND NOT i_steam_valve_stop_active THEN
    i_steam_valve_stop_active := TRUE;
    i_steam_valve_stop_scans := 0;
  END_IF;
  IF i_steam_valve_stop_active THEN
    i_steam_valve_stop_scans := i_steam_valve_stop_scans + 1;
    IF i_steam_valve_stop_scans >= 8 THEN
      steam_valve__coil__stop := FALSE;
      i_steam_valve_stop_active := FALSE;
      i_steam_valve_stop_scans := 0;
    END_IF;
  END_IF;
  IF steam_valve__coil__reset_trip AND NOT i_steam_valve_reset_trip_active THEN
    i_steam_valve_reset_trip_active := TRUE;
    i_steam_valve_reset_trip_scans := 0;
    IF steam_valve__holding__command_sequence >= 65535 THEN
      steam_valve__holding__command_sequence := 1;
    ELSE
      steam_valve__holding__command_sequence := steam_valve__holding__command_sequence + 1;
    END_IF;
    steam_valve__holding__reset_key := 42330;
  END_IF;
  IF i_steam_valve_reset_trip_active THEN
    i_steam_valve_reset_trip_scans := i_steam_valve_reset_trip_scans + 1;
    IF i_steam_valve_reset_trip_scans >= 8 THEN
      steam_valve__coil__reset_trip := FALSE;
      i_steam_valve_reset_trip_active := FALSE;
      i_steam_valve_reset_trip_scans := 0;
      steam_valve__holding__reset_key := 0;
    END_IF;
  END_IF;
  IF steam_valve__coil__ack_alarm AND NOT i_steam_valve_ack_alarm_active THEN
    i_steam_valve_ack_alarm_active := TRUE;
    i_steam_valve_ack_alarm_scans := 0;
  END_IF;
  IF i_steam_valve_ack_alarm_active THEN
    i_steam_valve_ack_alarm_scans := i_steam_valve_ack_alarm_scans + 1;
    IF i_steam_valve_ack_alarm_scans >= 8 THEN
      steam_valve__coil__ack_alarm := FALSE;
      i_steam_valve_ack_alarm_active := FALSE;
      i_steam_valve_ack_alarm_scans := 0;
    END_IF;
  END_IF;
  IF steam_valve__coil__trip_test AND NOT i_steam_valve_trip_test_active THEN
    i_steam_valve_trip_test_active := TRUE;
    i_steam_valve_trip_test_scans := 0;
  END_IF;
  IF i_steam_valve_trip_test_active THEN
    i_steam_valve_trip_test_scans := i_steam_valve_trip_test_scans + 1;
    IF i_steam_valve_trip_test_scans >= 8 THEN
      steam_valve__coil__trip_test := FALSE;
      i_steam_valve_trip_test_active := FALSE;
      i_steam_valve_trip_test_scans := 0;
    END_IF;
  END_IF;
  IF steam_valve__coil__clear_totalizer AND NOT i_steam_valve_clear_totalizer_active THEN
    i_steam_valve_clear_totalizer_active := TRUE;
    i_steam_valve_clear_totalizer_scans := 0;
  END_IF;
  IF i_steam_valve_clear_totalizer_active THEN
    i_steam_valve_clear_totalizer_scans := i_steam_valve_clear_totalizer_scans + 1;
    IF i_steam_valve_clear_totalizer_scans >= 8 THEN
      steam_valve__coil__clear_totalizer := FALSE;
      i_steam_valve_clear_totalizer_active := FALSE;
      i_steam_valve_clear_totalizer_scans := 0;
    END_IF;
  END_IF;
  IF turbine__coil__start AND NOT i_turbine_start_active THEN
    i_turbine_start_active := TRUE;
    i_turbine_start_scans := 0;
  END_IF;
  IF i_turbine_start_active THEN
    i_turbine_start_scans := i_turbine_start_scans + 1;
    IF i_turbine_start_scans >= 8 THEN
      turbine__coil__start := FALSE;
      i_turbine_start_active := FALSE;
      i_turbine_start_scans := 0;
    END_IF;
  END_IF;
  IF turbine__coil__stop AND NOT i_turbine_stop_active THEN
    i_turbine_stop_active := TRUE;
    i_turbine_stop_scans := 0;
  END_IF;
  IF i_turbine_stop_active THEN
    i_turbine_stop_scans := i_turbine_stop_scans + 1;
    IF i_turbine_stop_scans >= 8 THEN
      turbine__coil__stop := FALSE;
      i_turbine_stop_active := FALSE;
      i_turbine_stop_scans := 0;
    END_IF;
  END_IF;
  IF turbine__coil__reset_trip AND NOT i_turbine_reset_trip_active THEN
    i_turbine_reset_trip_active := TRUE;
    i_turbine_reset_trip_scans := 0;
    IF turbine__holding__command_sequence >= 65535 THEN
      turbine__holding__command_sequence := 1;
    ELSE
      turbine__holding__command_sequence := turbine__holding__command_sequence + 1;
    END_IF;
    turbine__holding__reset_key := 42330;
  END_IF;
  IF i_turbine_reset_trip_active THEN
    i_turbine_reset_trip_scans := i_turbine_reset_trip_scans + 1;
    IF i_turbine_reset_trip_scans >= 8 THEN
      turbine__coil__reset_trip := FALSE;
      i_turbine_reset_trip_active := FALSE;
      i_turbine_reset_trip_scans := 0;
      turbine__holding__reset_key := 0;
    END_IF;
  END_IF;
  IF turbine__coil__ack_alarm AND NOT i_turbine_ack_alarm_active THEN
    i_turbine_ack_alarm_active := TRUE;
    i_turbine_ack_alarm_scans := 0;
  END_IF;
  IF i_turbine_ack_alarm_active THEN
    i_turbine_ack_alarm_scans := i_turbine_ack_alarm_scans + 1;
    IF i_turbine_ack_alarm_scans >= 8 THEN
      turbine__coil__ack_alarm := FALSE;
      i_turbine_ack_alarm_active := FALSE;
      i_turbine_ack_alarm_scans := 0;
    END_IF;
  END_IF;
  IF turbine__coil__trip_test AND NOT i_turbine_trip_test_active THEN
    i_turbine_trip_test_active := TRUE;
    i_turbine_trip_test_scans := 0;
  END_IF;
  IF i_turbine_trip_test_active THEN
    i_turbine_trip_test_scans := i_turbine_trip_test_scans + 1;
    IF i_turbine_trip_test_scans >= 8 THEN
      turbine__coil__trip_test := FALSE;
      i_turbine_trip_test_active := FALSE;
      i_turbine_trip_test_scans := 0;
    END_IF;
  END_IF;
  IF turbine__coil__clear_totalizer AND NOT i_turbine_clear_totalizer_active THEN
    i_turbine_clear_totalizer_active := TRUE;
    i_turbine_clear_totalizer_scans := 0;
  END_IF;
  IF i_turbine_clear_totalizer_active THEN
    i_turbine_clear_totalizer_scans := i_turbine_clear_totalizer_scans + 1;
    IF i_turbine_clear_totalizer_scans >= 8 THEN
      turbine__coil__clear_totalizer := FALSE;
      i_turbine_clear_totalizer_active := FALSE;
      i_turbine_clear_totalizer_scans := 0;
    END_IF;
  END_IF;
  IF generator__coil__start AND NOT i_generator_start_active THEN
    i_generator_start_active := TRUE;
    i_generator_start_scans := 0;
  END_IF;
  IF i_generator_start_active THEN
    i_generator_start_scans := i_generator_start_scans + 1;
    IF i_generator_start_scans >= 8 THEN
      generator__coil__start := FALSE;
      i_generator_start_active := FALSE;
      i_generator_start_scans := 0;
    END_IF;
  END_IF;
  IF generator__coil__stop AND NOT i_generator_stop_active THEN
    i_generator_stop_active := TRUE;
    i_generator_stop_scans := 0;
  END_IF;
  IF i_generator_stop_active THEN
    i_generator_stop_scans := i_generator_stop_scans + 1;
    IF i_generator_stop_scans >= 8 THEN
      generator__coil__stop := FALSE;
      i_generator_stop_active := FALSE;
      i_generator_stop_scans := 0;
    END_IF;
  END_IF;
  IF generator__coil__reset_trip AND NOT i_generator_reset_trip_active THEN
    i_generator_reset_trip_active := TRUE;
    i_generator_reset_trip_scans := 0;
    IF generator__holding__command_sequence >= 65535 THEN
      generator__holding__command_sequence := 1;
    ELSE
      generator__holding__command_sequence := generator__holding__command_sequence + 1;
    END_IF;
    generator__holding__reset_key := 42330;
  END_IF;
  IF i_generator_reset_trip_active THEN
    i_generator_reset_trip_scans := i_generator_reset_trip_scans + 1;
    IF i_generator_reset_trip_scans >= 8 THEN
      generator__coil__reset_trip := FALSE;
      i_generator_reset_trip_active := FALSE;
      i_generator_reset_trip_scans := 0;
      generator__holding__reset_key := 0;
    END_IF;
  END_IF;
  IF generator__coil__ack_alarm AND NOT i_generator_ack_alarm_active THEN
    i_generator_ack_alarm_active := TRUE;
    i_generator_ack_alarm_scans := 0;
  END_IF;
  IF i_generator_ack_alarm_active THEN
    i_generator_ack_alarm_scans := i_generator_ack_alarm_scans + 1;
    IF i_generator_ack_alarm_scans >= 8 THEN
      generator__coil__ack_alarm := FALSE;
      i_generator_ack_alarm_active := FALSE;
      i_generator_ack_alarm_scans := 0;
    END_IF;
  END_IF;
  IF generator__coil__trip_test AND NOT i_generator_trip_test_active THEN
    i_generator_trip_test_active := TRUE;
    i_generator_trip_test_scans := 0;
  END_IF;
  IF i_generator_trip_test_active THEN
    i_generator_trip_test_scans := i_generator_trip_test_scans + 1;
    IF i_generator_trip_test_scans >= 8 THEN
      generator__coil__trip_test := FALSE;
      i_generator_trip_test_active := FALSE;
      i_generator_trip_test_scans := 0;
    END_IF;
  END_IF;
  IF generator__coil__clear_totalizer AND NOT i_generator_clear_totalizer_active THEN
    i_generator_clear_totalizer_active := TRUE;
    i_generator_clear_totalizer_scans := 0;
  END_IF;
  IF i_generator_clear_totalizer_active THEN
    i_generator_clear_totalizer_scans := i_generator_clear_totalizer_scans + 1;
    IF i_generator_clear_totalizer_scans >= 8 THEN
      generator__coil__clear_totalizer := FALSE;
      i_generator_clear_totalizer_active := FALSE;
      i_generator_clear_totalizer_scans := 0;
    END_IF;
  END_IF;
  IF generator__coil__breaker_close AND NOT i_generator_breaker_close_active THEN
    i_generator_breaker_close_active := TRUE;
    i_generator_breaker_close_scans := 0;
  END_IF;
  IF i_generator_breaker_close_active THEN
    i_generator_breaker_close_scans := i_generator_breaker_close_scans + 1;
    IF i_generator_breaker_close_scans >= 8 THEN
      generator__coil__breaker_close := FALSE;
      i_generator_breaker_close_active := FALSE;
      i_generator_breaker_close_scans := 0;
    END_IF;
  END_IF;
  IF generator__coil__breaker_open AND NOT i_generator_breaker_open_active THEN
    i_generator_breaker_open_active := TRUE;
    i_generator_breaker_open_scans := 0;
  END_IF;
  IF i_generator_breaker_open_active THEN
    i_generator_breaker_open_scans := i_generator_breaker_open_scans + 1;
    IF i_generator_breaker_open_scans >= 8 THEN
      generator__coil__breaker_open := FALSE;
      i_generator_breaker_open_active := FALSE;
      i_generator_breaker_open_scans := 0;
    END_IF;
  END_IF;
